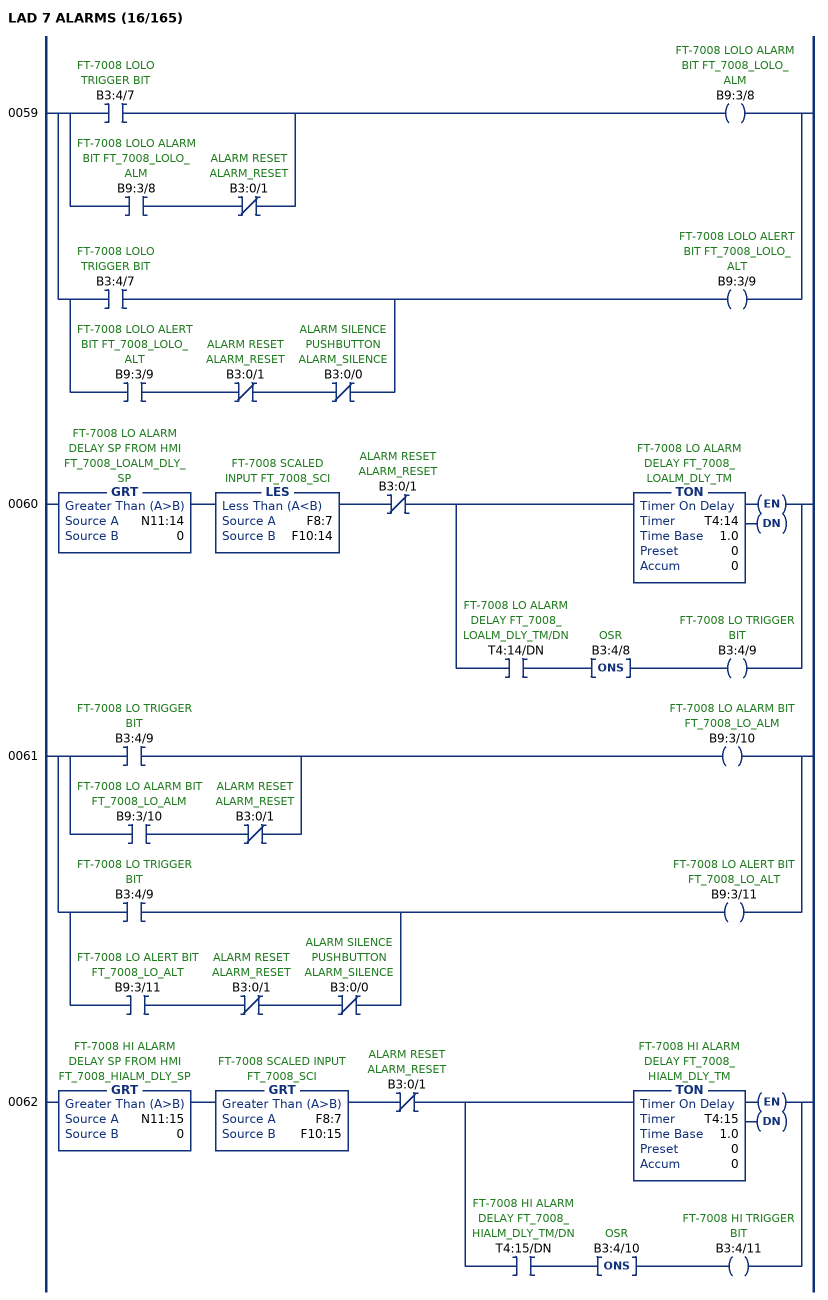
% Rung: 59 %
SOR BST BST XIC B3:4/7 NXB XIC B9:3/8 XIO B3:0/1 BND OTE B9:3/8 NXB BST XIC B3:4/7 NXB XIC B9:3/9 XIO B3:0/1 XIO B3:0/0 BND OTE B9:3/9 BND EOR
%   B3:4/7  "FT-7008 LOLO TRIGGER BIT" %
%   B9:3/8  FT_7008_LOLO_ALM  "FT-7008 LOLO ALARM BIT" %
%   B3:0/1  ALARM_RESET  "ALARM RESET" %
%   B9:3/9  FT_7008_LOLO_ALT  "FT-7008 LOLO ALERT BIT" %
%   B3:0/0  ALARM_SILENCE  "ALARM SILENCE PUSHBUTTON" %
% Rung: 60 %
SOR GRT N11:14 0 LES F8:7 F10:14 XIO B3:0/1 BST TON T4:14 1.0 0 0 NXB XIC T4:14/DN OSR B3:4/8 OTE B3:4/9 BND EOR
%   N11:14  FT_7008_LOALM_DLY_SP  "FT-7008 LO ALARM DELAY SP FROM HMI" %
%   F8:7  FT_7008_SCI  "FT-7008 SCALED INPUT" %
%   F10:14  FT_7008_LOALM_SP  "FT-7008 LO ALARM SP" %
%   B3:0/1  ALARM_RESET  "ALARM RESET" %
%   T4:14  FT_7008_LOALM_DLY_TM  "FT-7008 LO ALARM DELAY" %
%   B3:4/8  "OSR" %
%   B3:4/9  "FT-7008 LO TRIGGER BIT" %
% Rung: 61 %
SOR BST BST XIC B3:4/9 NXB XIC B9:3/10 XIO B3:0/1 BND OTE B9:3/10 NXB BST XIC B3:4/9 NXB XIC B9:3/11 XIO B3:0/1 XIO B3:0/0 BND OTE B9:3/11 BND EOR
%   B3:4/9  "FT-7008 LO TRIGGER BIT" %
%   B9:3/10  FT_7008_LO_ALM  "FT-7008 LO ALARM BIT" %
%   B3:0/1  ALARM_RESET  "ALARM RESET" %
%   B9:3/11  FT_7008_LO_ALT  "FT-7008 LO ALERT BIT" %
%   B3:0/0  ALARM_SILENCE  "ALARM SILENCE PUSHBUTTON" %
% Rung: 62 %
SOR GRT N11:15 0 GRT F8:7 F10:15 XIO B3:0/1 BST TON T4:15 1.0 0 0 NXB XIC T4:15/DN OSR B3:4/10 OTE B3:4/11 BND EOR
%   N11:15  FT_7008_HIALM_DLY_SP  "FT-7008 HI ALARM DELAY SP FROM HMI" %
%   F8:7  FT_7008_SCI  "FT-7008 SCALED INPUT" %
%   F10:15  FT_7008_HIALM_SP  "FT-7008 HI ALARM SP" %
%   B3:0/1  ALARM_RESET  "ALARM RESET" %
%   T4:15  FT_7008_HIALM_DLY_TM  "FT-7008 HI ALARM DELAY" %
%   B3:4/10  "OSR" %
%   B3:4/11  "FT-7008 HI TRIGGER BIT" %

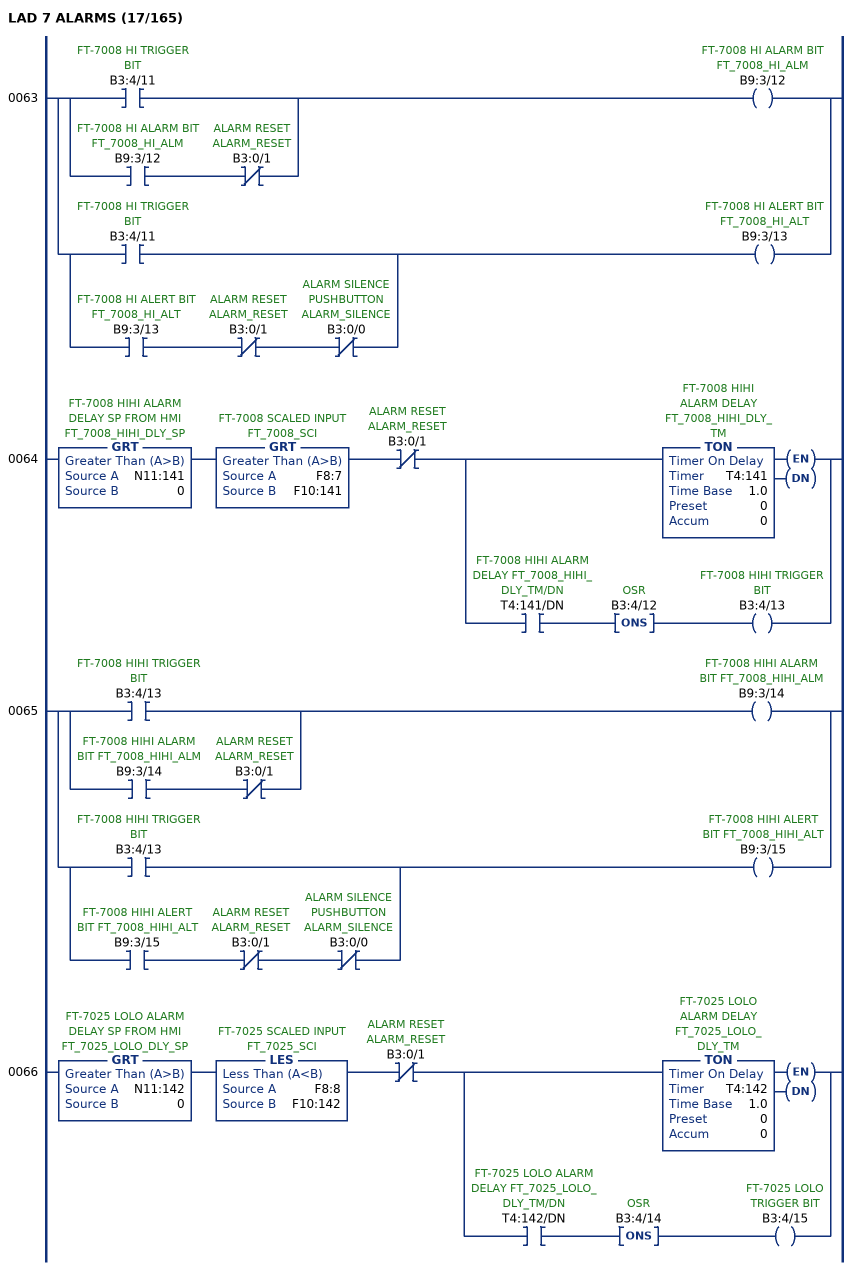
% Rung: 63 %
SOR BST BST XIC B3:4/11 NXB XIC B9:3/12 XIO B3:0/1 BND OTE B9:3/12 NXB BST XIC B3:4/11 NXB XIC B9:3/13 XIO B3:0/1 XIO B3:0/0 BND OTE B9:3/13 BND EOR
%   B3:4/11  "FT-7008 HI TRIGGER BIT" %
%   B9:3/12  FT_7008_HI_ALM  "FT-7008 HI ALARM BIT" %
%   B3:0/1  ALARM_RESET  "ALARM RESET" %
%   B9:3/13  FT_7008_HI_ALT  "FT-7008 HI ALERT BIT" %
%   B3:0/0  ALARM_SILENCE  "ALARM SILENCE PUSHBUTTON" %
% Rung: 64 %
SOR GRT N11:141 0 GRT F8:7 F10:141 XIO B3:0/1 BST TON T4:141 1.0 0 0 NXB XIC T4:141/DN OSR B3:4/12 OTE B3:4/13 BND EOR
%   N11:141  FT_7008_HIHI_DLY_SP  "FT-7008 HIHI ALARM DELAY SP FROM HMI" %
%   F8:7  FT_7008_SCI  "FT-7008 SCALED INPUT" %
%   F10:141  FT_7008_HIHI_SP  "FT-7008 HIHI ALARM SP" %
%   B3:0/1  ALARM_RESET  "ALARM RESET" %
%   T4:141  FT_7008_HIHI_DLY_TM  "FT-7008 HIHI ALARM DELAY" %
%   B3:4/12  "OSR" %
%   B3:4/13  "FT-7008 HIHI TRIGGER BIT" %
% Rung: 65 %
SOR BST BST XIC B3:4/13 NXB XIC B9:3/14 XIO B3:0/1 BND OTE B9:3/14 NXB BST XIC B3:4/13 NXB XIC B9:3/15 XIO B3:0/1 XIO B3:0/0 BND OTE B9:3/15 BND EOR
%   B3:4/13  "FT-7008 HIHI TRIGGER BIT" %
%   B9:3/14  FT_7008_HIHI_ALM  "FT-7008 HIHI ALARM BIT" %
%   B3:0/1  ALARM_RESET  "ALARM RESET" %
%   B9:3/15  FT_7008_HIHI_ALT  "FT-7008 HIHI ALERT BIT" %
%   B3:0/0  ALARM_SILENCE  "ALARM SILENCE PUSHBUTTON" %
% Rung: 66 %
SOR GRT N11:142 0 LES F8:8 F10:142 XIO B3:0/1 BST TON T4:142 1.0 0 0 NXB XIC T4:142/DN OSR B3:4/14 OTE B3:4/15 BND EOR
%   N11:142  FT_7025_LOLO_DLY_SP  "FT-7025 LOLO ALARM DELAY SP FROM HMI" %
%   F8:8  FT_7025_SCI  "FT-7025 SCALED INPUT" %
%   F10:142  FT_7025_LOLO_SP  "FT-7025 LOLO ALARM SP" %
%   B3:0/1  ALARM_RESET  "ALARM RESET" %
%   T4:142  FT_7025_LOLO_DLY_TM  "FT-7025 LOLO ALARM DELAY" %
%   B3:4/14  "OSR" %
%   B3:4/15  "FT-7025 LOLO TRIGGER BIT" %

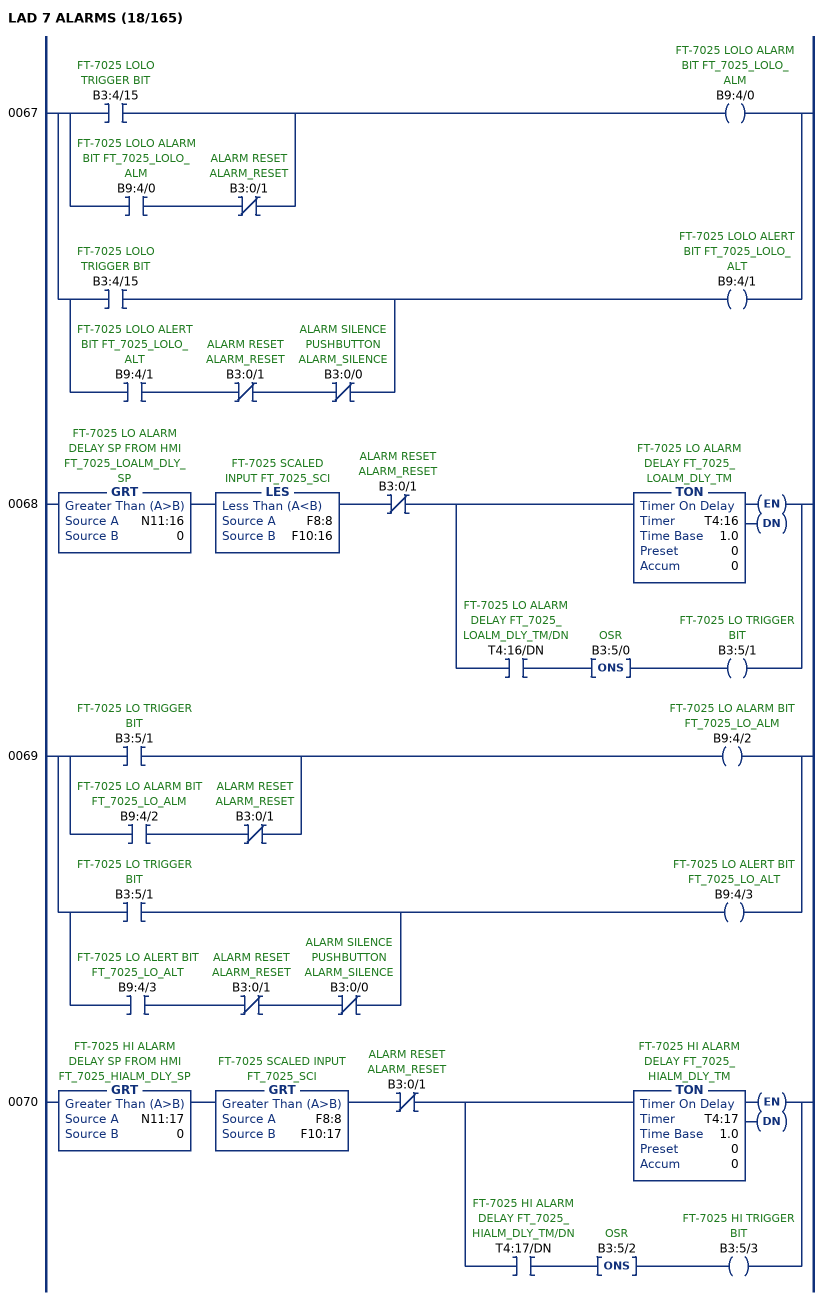
% Rung: 67 %
SOR BST BST XIC B3:4/15 NXB XIC B9:4/0 XIO B3:0/1 BND OTE B9:4/0 NXB BST XIC B3:4/15 NXB XIC B9:4/1 XIO B3:0/1 XIO B3:0/0 BND OTE B9:4/1 BND EOR
%   B3:4/15  "FT-7025 LOLO TRIGGER BIT" %
%   B9:4/0  FT_7025_LOLO_ALM  "FT-7025 LOLO ALARM BIT" %
%   B3:0/1  ALARM_RESET  "ALARM RESET" %
%   B9:4/1  FT_7025_LOLO_ALT  "FT-7025 LOLO ALERT BIT" %
%   B3:0/0  ALARM_SILENCE  "ALARM SILENCE PUSHBUTTON" %
% Rung: 68 %
SOR GRT N11:16 0 LES F8:8 F10:16 XIO B3:0/1 BST TON T4:16 1.0 0 0 NXB XIC T4:16/DN OSR B3:5/0 OTE B3:5/1 BND EOR
%   N11:16  FT_7025_LOALM_DLY_SP  "FT-7025 LO ALARM DELAY SP FROM HMI" %
%   F8:8  FT_7025_SCI  "FT-7025 SCALED INPUT" %
%   F10:16  FT_7025_LOALM_SP  "FT-7025 LO ALARM SP" %
%   B3:0/1  ALARM_RESET  "ALARM RESET" %
%   T4:16  FT_7025_LOALM_DLY_TM  "FT-7025 LO ALARM DELAY" %
%   B3:5/0  "OSR" %
%   B3:5/1  "FT-7025 LO TRIGGER BIT" %
% Rung: 69 %
SOR BST BST XIC B3:5/1 NXB XIC B9:4/2 XIO B3:0/1 BND OTE B9:4/2 NXB BST XIC B3:5/1 NXB XIC B9:4/3 XIO B3:0/1 XIO B3:0/0 BND OTE B9:4/3 BND EOR
%   B3:5/1  "FT-7025 LO TRIGGER BIT" %
%   B9:4/2  FT_7025_LO_ALM  "FT-7025 LO ALARM BIT" %
%   B3:0/1  ALARM_RESET  "ALARM RESET" %
%   B9:4/3  FT_7025_LO_ALT  "FT-7025 LO ALERT BIT" %
%   B3:0/0  ALARM_SILENCE  "ALARM SILENCE PUSHBUTTON" %
% Rung: 70 %
SOR GRT N11:17 0 GRT F8:8 F10:17 XIO B3:0/1 BST TON T4:17 1.0 0 0 NXB XIC T4:17/DN OSR B3:5/2 OTE B3:5/3 BND EOR
%   N11:17  FT_7025_HIALM_DLY_SP  "FT-7025 HI ALARM DELAY SP FROM HMI" %
%   F8:8  FT_7025_SCI  "FT-7025 SCALED INPUT" %
%   F10:17  FT_7025_HIALM_SP  "FT-7025 HI ALARM SP" %
%   B3:0/1  ALARM_RESET  "ALARM RESET" %
%   T4:17  FT_7025_HIALM_DLY_TM  "FT-7025 HI ALARM DELAY" %
%   B3:5/2  "OSR" %
%   B3:5/3  "FT-7025 HI TRIGGER BIT" %

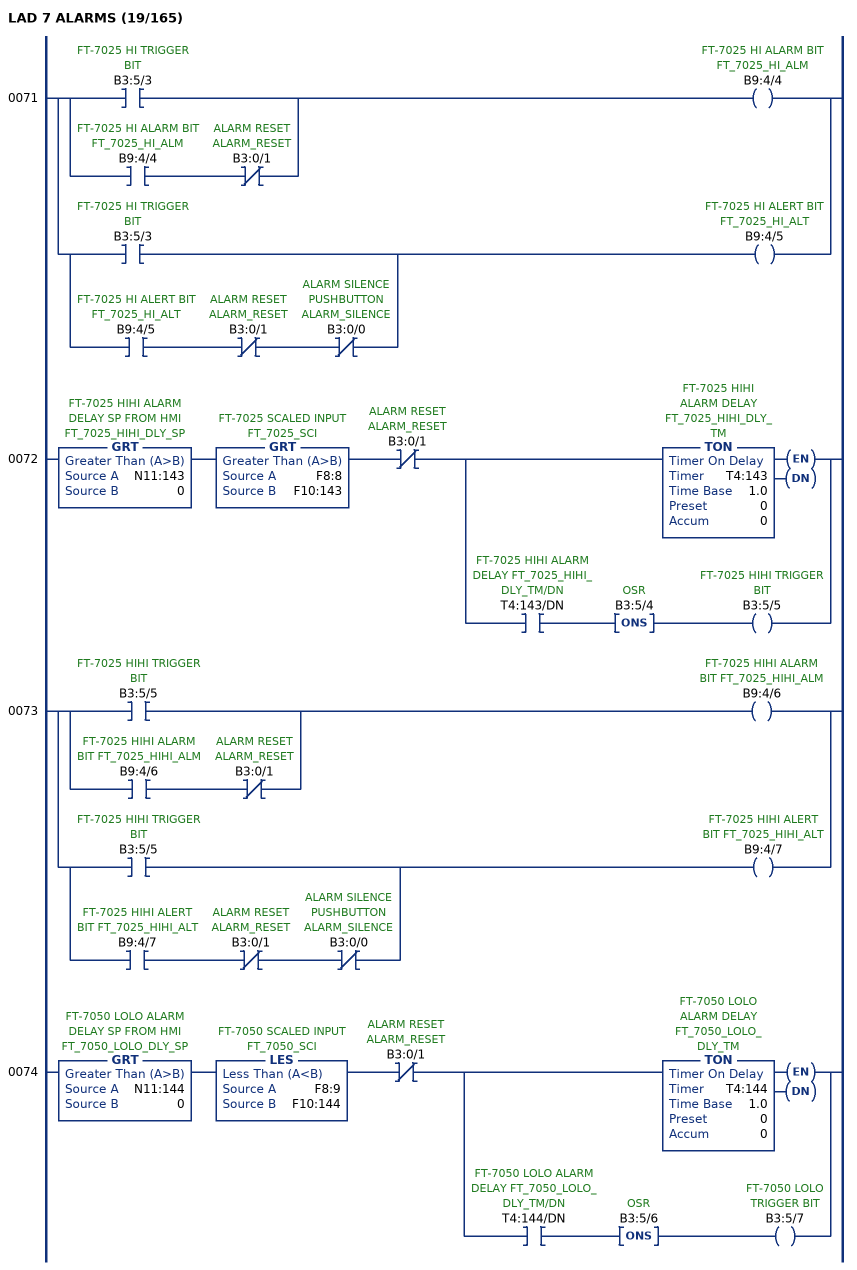
% Rung: 71 %
SOR BST BST XIC B3:5/3 NXB XIC B9:4/4 XIO B3:0/1 BND OTE B9:4/4 NXB BST XIC B3:5/3 NXB XIC B9:4/5 XIO B3:0/1 XIO B3:0/0 BND OTE B9:4/5 BND EOR
%   B3:5/3  "FT-7025 HI TRIGGER BIT" %
%   B9:4/4  FT_7025_HI_ALM  "FT-7025 HI ALARM BIT" %
%   B3:0/1  ALARM_RESET  "ALARM RESET" %
%   B9:4/5  FT_7025_HI_ALT  "FT-7025 HI ALERT BIT" %
%   B3:0/0  ALARM_SILENCE  "ALARM SILENCE PUSHBUTTON" %
% Rung: 72 %
SOR GRT N11:143 0 GRT F8:8 F10:143 XIO B3:0/1 BST TON T4:143 1.0 0 0 NXB XIC T4:143/DN OSR B3:5/4 OTE B3:5/5 BND EOR
%   N11:143  FT_7025_HIHI_DLY_SP  "FT-7025 HIHI ALARM DELAY SP FROM HMI" %
%   F8:8  FT_7025_SCI  "FT-7025 SCALED INPUT" %
%   F10:143  FT_7025_HIHI_SP  "FT-7025 HIHI ALARM SP" %
%   B3:0/1  ALARM_RESET  "ALARM RESET" %
%   T4:143  FT_7025_HIHI_DLY_TM  "FT-7025 HIHI ALARM DELAY" %
%   B3:5/4  "OSR" %
%   B3:5/5  "FT-7025 HIHI TRIGGER BIT" %
% Rung: 73 %
SOR BST BST XIC B3:5/5 NXB XIC B9:4/6 XIO B3:0/1 BND OTE B9:4/6 NXB BST XIC B3:5/5 NXB XIC B9:4/7 XIO B3:0/1 XIO B3:0/0 BND OTE B9:4/7 BND EOR
%   B3:5/5  "FT-7025 HIHI TRIGGER BIT" %
%   B9:4/6  FT_7025_HIHI_ALM  "FT-7025 HIHI ALARM BIT" %
%   B3:0/1  ALARM_RESET  "ALARM RESET" %
%   B9:4/7  FT_7025_HIHI_ALT  "FT-7025 HIHI ALERT BIT" %
%   B3:0/0  ALARM_SILENCE  "ALARM SILENCE PUSHBUTTON" %
% Rung: 74 %
SOR GRT N11:144 0 LES F8:9 F10:144 XIO B3:0/1 BST TON T4:144 1.0 0 0 NXB XIC T4:144/DN OSR B3:5/6 OTE B3:5/7 BND EOR
%   N11:144  FT_7050_LOLO_DLY_SP  "FT-7050 LOLO ALARM DELAY SP FROM HMI" %
%   F8:9  FT_7050_SCI  "FT-7050 SCALED INPUT" %
%   F10:144  FT_7050_LOLO_SP  "FT-7050 LOLO ALARM SP" %
%   B3:0/1  ALARM_RESET  "ALARM RESET" %
%   T4:144  FT_7050_LOLO_DLY_TM  "FT-7050 LOLO ALARM DELAY" %
%   B3:5/6  "OSR" %
%   B3:5/7  "FT-7050 LOLO TRIGGER BIT" %

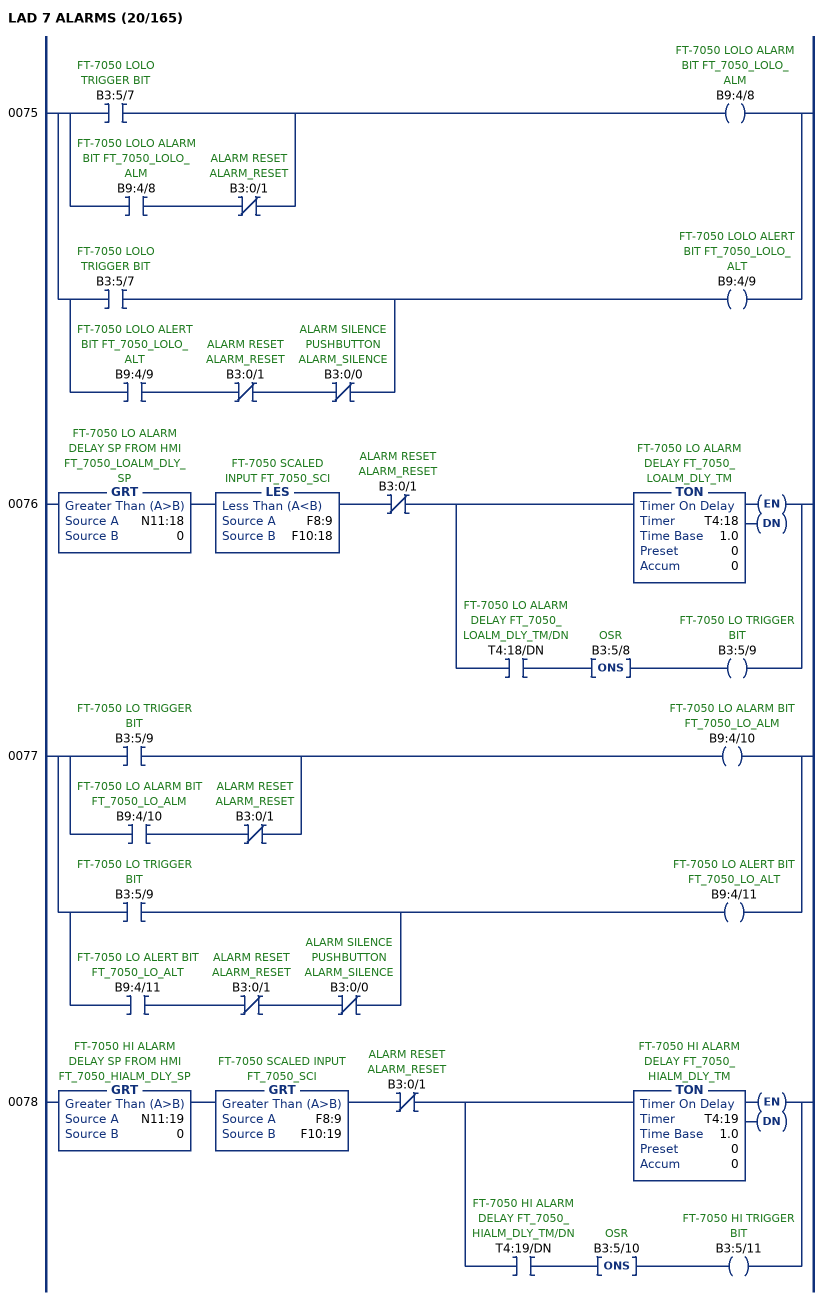
% Rung: 75 %
SOR BST BST XIC B3:5/7 NXB XIC B9:4/8 XIO B3:0/1 BND OTE B9:4/8 NXB BST XIC B3:5/7 NXB XIC B9:4/9 XIO B3:0/1 XIO B3:0/0 BND OTE B9:4/9 BND EOR
%   B3:5/7  "FT-7050 LOLO TRIGGER BIT" %
%   B9:4/8  FT_7050_LOLO_ALM  "FT-7050 LOLO ALARM BIT" %
%   B3:0/1  ALARM_RESET  "ALARM RESET" %
%   B9:4/9  FT_7050_LOLO_ALT  "FT-7050 LOLO ALERT BIT" %
%   B3:0/0  ALARM_SILENCE  "ALARM SILENCE PUSHBUTTON" %
% Rung: 76 %
SOR GRT N11:18 0 LES F8:9 F10:18 XIO B3:0/1 BST TON T4:18 1.0 0 0 NXB XIC T4:18/DN OSR B3:5/8 OTE B3:5/9 BND EOR
%   N11:18  FT_7050_LOALM_DLY_SP  "FT-7050 LO ALARM DELAY SP FROM HMI" %
%   F8:9  FT_7050_SCI  "FT-7050 SCALED INPUT" %
%   F10:18  FT_7050_LOALM_SP  "FT-7050 LO ALARM SP" %
%   B3:0/1  ALARM_RESET  "ALARM RESET" %
%   T4:18  FT_7050_LOALM_DLY_TM  "FT-7050 LO ALARM DELAY" %
%   B3:5/8  "OSR" %
%   B3:5/9  "FT-7050 LO TRIGGER BIT" %
% Rung: 77 %
SOR BST BST XIC B3:5/9 NXB XIC B9:4/10 XIO B3:0/1 BND OTE B9:4/10 NXB BST XIC B3:5/9 NXB XIC B9:4/11 XIO B3:0/1 XIO B3:0/0 BND OTE B9:4/11 BND EOR
%   B3:5/9  "FT-7050 LO TRIGGER BIT" %
%   B9:4/10  FT_7050_LO_ALM  "FT-7050 LO ALARM BIT" %
%   B3:0/1  ALARM_RESET  "ALARM RESET" %
%   B9:4/11  FT_7050_LO_ALT  "FT-7050 LO ALERT BIT" %
%   B3:0/0  ALARM_SILENCE  "ALARM SILENCE PUSHBUTTON" %
% Rung: 78 %
SOR GRT N11:19 0 GRT F8:9 F10:19 XIO B3:0/1 BST TON T4:19 1.0 0 0 NXB XIC T4:19/DN OSR B3:5/10 OTE B3:5/11 BND EOR
%   N11:19  FT_7050_HIALM_DLY_SP  "FT-7050 HI ALARM DELAY SP FROM HMI" %
%   F8:9  FT_7050_SCI  "FT-7050 SCALED INPUT" %
%   F10:19  FT_7050_HIALM_SP  "FT-7050 HI ALARM SP" %
%   B3:0/1  ALARM_RESET  "ALARM RESET" %
%   T4:19  FT_7050_HIALM_DLY_TM  "FT-7050 HI ALARM DELAY" %
%   B3:5/10  "OSR" %
%   B3:5/11  "FT-7050 HI TRIGGER BIT" %

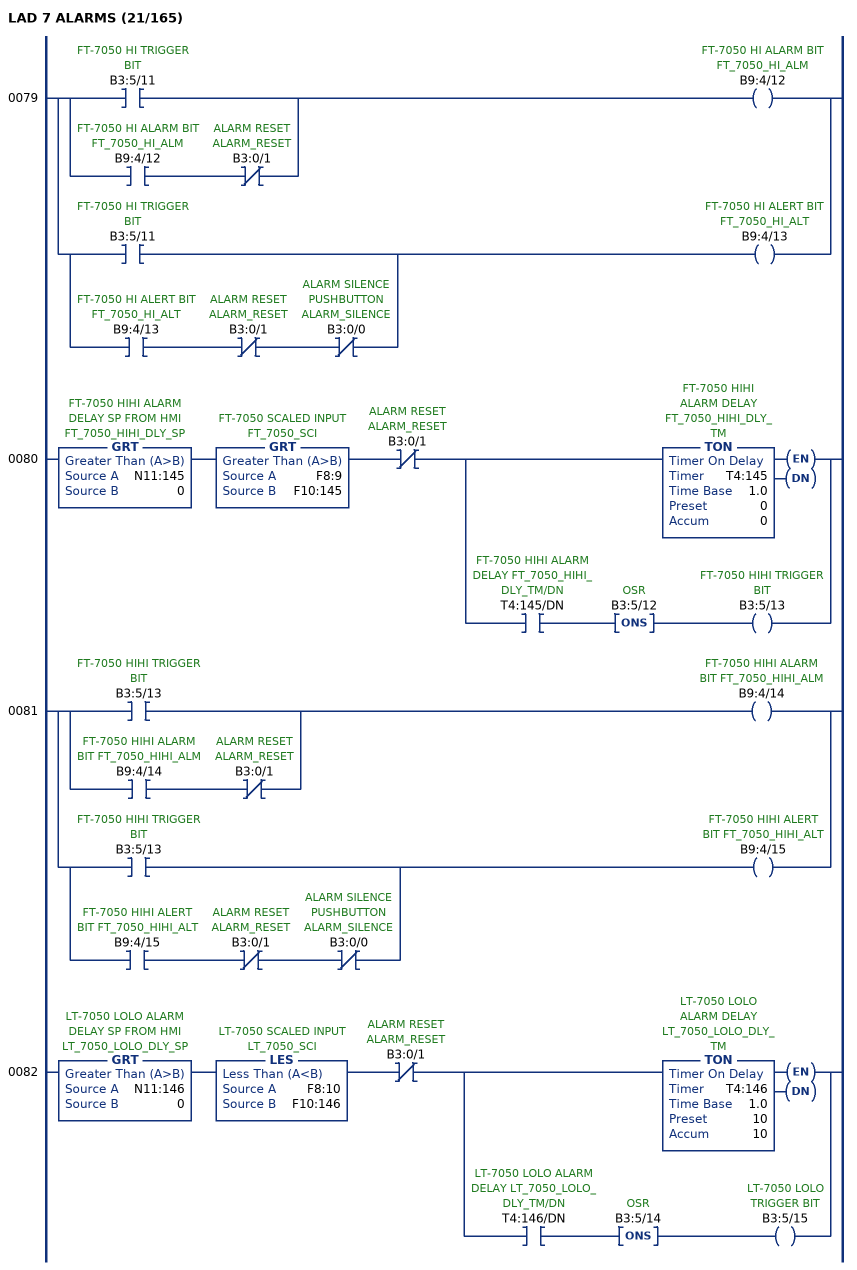
% Rung: 79 %
SOR BST BST XIC B3:5/11 NXB XIC B9:4/12 XIO B3:0/1 BND OTE B9:4/12 NXB BST XIC B3:5/11 NXB XIC B9:4/13 XIO B3:0/1 XIO B3:0/0 BND OTE B9:4/13 BND EOR
%   B3:5/11  "FT-7050 HI TRIGGER BIT" %
%   B9:4/12  FT_7050_HI_ALM  "FT-7050 HI ALARM BIT" %
%   B3:0/1  ALARM_RESET  "ALARM RESET" %
%   B9:4/13  FT_7050_HI_ALT  "FT-7050 HI ALERT BIT" %
%   B3:0/0  ALARM_SILENCE  "ALARM SILENCE PUSHBUTTON" %
% Rung: 80 %
SOR GRT N11:145 0 GRT F8:9 F10:145 XIO B3:0/1 BST TON T4:145 1.0 0 0 NXB XIC T4:145/DN OSR B3:5/12 OTE B3:5/13 BND EOR
%   N11:145  FT_7050_HIHI_DLY_SP  "FT-7050 HIHI ALARM DELAY SP FROM HMI" %
%   F8:9  FT_7050_SCI  "FT-7050 SCALED INPUT" %
%   F10:145  FT_7050_HIHI_SP  "FT-7050 HIHI ALARM SP" %
%   B3:0/1  ALARM_RESET  "ALARM RESET" %
%   T4:145  FT_7050_HIHI_DLY_TM  "FT-7050 HIHI ALARM DELAY" %
%   B3:5/12  "OSR" %
%   B3:5/13  "FT-7050 HIHI TRIGGER BIT" %
% Rung: 81 %
SOR BST BST XIC B3:5/13 NXB XIC B9:4/14 XIO B3:0/1 BND OTE B9:4/14 NXB BST XIC B3:5/13 NXB XIC B9:4/15 XIO B3:0/1 XIO B3:0/0 BND OTE B9:4/15 BND EOR
%   B3:5/13  "FT-7050 HIHI TRIGGER BIT" %
%   B9:4/14  FT_7050_HIHI_ALM  "FT-7050 HIHI ALARM BIT" %
%   B3:0/1  ALARM_RESET  "ALARM RESET" %
%   B9:4/15  FT_7050_HIHI_ALT  "FT-7050 HIHI ALERT BIT" %
%   B3:0/0  ALARM_SILENCE  "ALARM SILENCE PUSHBUTTON" %
% Rung: 82 %
SOR GRT N11:146 0 LES F8:10 F10:146 XIO B3:0/1 BST TON T4:146 1.0 10 10 NXB XIC T4:146/DN OSR B3:5/14 OTE B3:5/15 BND EOR
%   N11:146  LT_7050_LOLO_DLY_SP  "LT-7050 LOLO ALARM DELAY SP FROM HMI" %
%   F8:10  LT_7050_SCI  "LT-7050 SCALED INPUT" %
%   F10:146  LT_7050_LOLO_SP  "LT-7050 LOLO ALARM SP" %
%   B3:0/1  ALARM_RESET  "ALARM RESET" %
%   T4:146  LT_7050_LOLO_DLY_TM  "LT-7050 LOLO ALARM DELAY" %
%   B3:5/14  "OSR" %
%   B3:5/15  "LT-7050 LOLO TRIGGER BIT" %

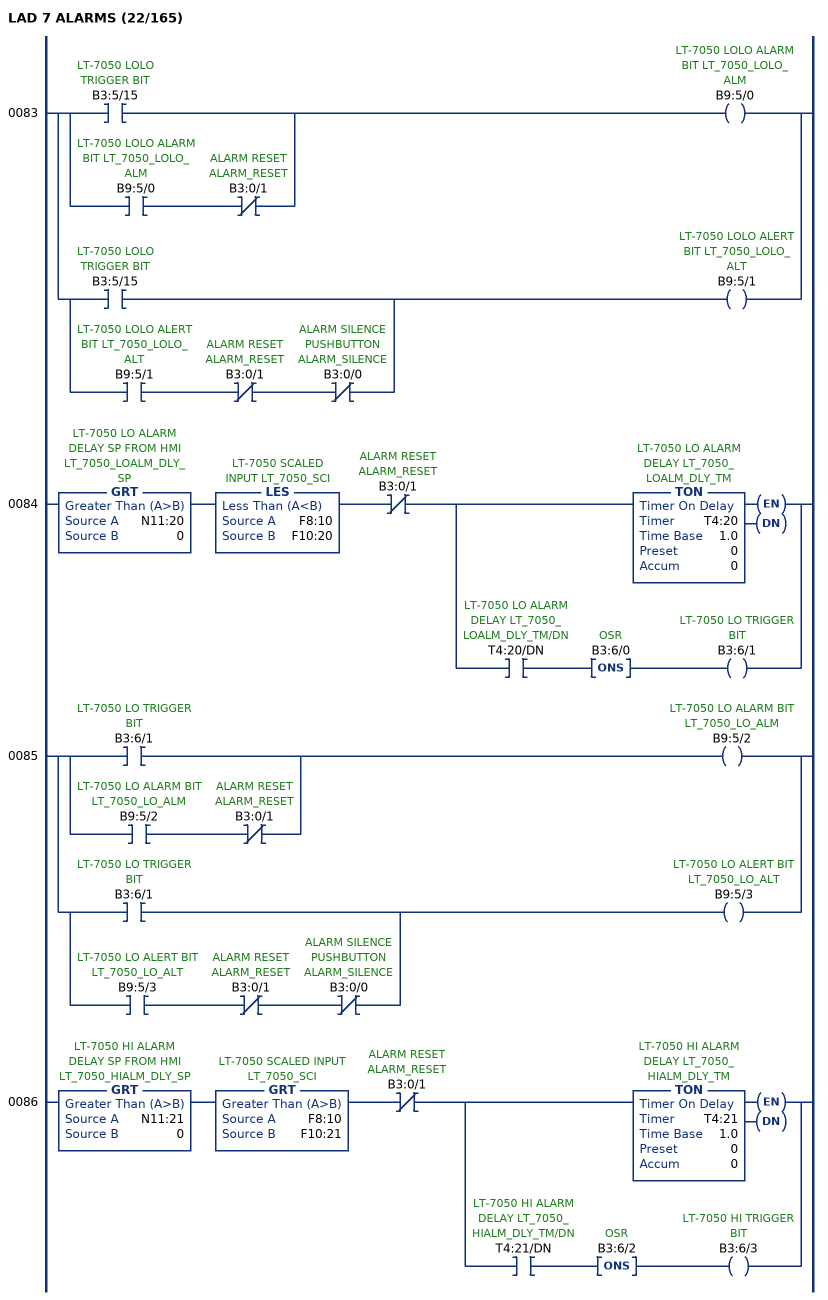
% Rung: 83 %
SOR BST BST XIC B3:5/15 NXB XIC B9:5/0 XIO B3:0/1 BND OTE B9:5/0 NXB BST XIC B3:5/15 NXB XIC B9:5/1 XIO B3:0/1 XIO B3:0/0 BND OTE B9:5/1 BND EOR
%   B3:5/15  "LT-7050 LOLO TRIGGER BIT" %
%   B9:5/0  LT_7050_LOLO_ALM  "LT-7050 LOLO ALARM BIT" %
%   B3:0/1  ALARM_RESET  "ALARM RESET" %
%   B9:5/1  LT_7050_LOLO_ALT  "LT-7050 LOLO ALERT BIT" %
%   B3:0/0  ALARM_SILENCE  "ALARM SILENCE PUSHBUTTON" %
% Rung: 84 %
SOR GRT N11:20 0 LES F8:10 F10:20 XIO B3:0/1 BST TON T4:20 1.0 0 0 NXB XIC T4:20/DN OSR B3:6/0 OTE B3:6/1 BND EOR
%   N11:20  LT_7050_LOALM_DLY_SP  "LT-7050 LO ALARM DELAY SP FROM HMI" %
%   F8:10  LT_7050_SCI  "LT-7050 SCALED INPUT" %
%   F10:20  LT_7050_LOALM_SP  "LT-7050 LO ALARM SP" %
%   B3:0/1  ALARM_RESET  "ALARM RESET" %
%   T4:20  LT_7050_LOALM_DLY_TM  "LT-7050 LO ALARM DELAY" %
%   B3:6/0  "OSR" %
%   B3:6/1  "LT-7050 LO TRIGGER BIT" %
% Rung: 85 %
SOR BST BST XIC B3:6/1 NXB XIC B9:5/2 XIO B3:0/1 BND OTE B9:5/2 NXB BST XIC B3:6/1 NXB XIC B9:5/3 XIO B3:0/1 XIO B3:0/0 BND OTE B9:5/3 BND EOR
%   B3:6/1  "LT-7050 LO TRIGGER BIT" %
%   B9:5/2  LT_7050_LO_ALM  "LT-7050 LO ALARM BIT" %
%   B3:0/1  ALARM_RESET  "ALARM RESET" %
%   B9:5/3  LT_7050_LO_ALT  "LT-7050 LO ALERT BIT" %
%   B3:0/0  ALARM_SILENCE  "ALARM SILENCE PUSHBUTTON" %
% Rung: 86 %
SOR GRT N11:21 0 GRT F8:10 F10:21 XIO B3:0/1 BST TON T4:21 1.0 0 0 NXB XIC T4:21/DN OSR B3:6/2 OTE B3:6/3 BND EOR
%   N11:21  LT_7050_HIALM_DLY_SP  "LT-7050 HI ALARM DELAY SP FROM HMI" %
%   F8:10  LT_7050_SCI  "LT-7050 SCALED INPUT" %
%   F10:21  LT_7050_HIALM_SP  "LT-7050 HI ALARM SP" %
%   B3:0/1  ALARM_RESET  "ALARM RESET" %
%   T4:21  LT_7050_HIALM_DLY_TM  "LT-7050 HI ALARM DELAY" %
%   B3:6/2  "OSR" %
%   B3:6/3  "LT-7050 HI TRIGGER BIT" %

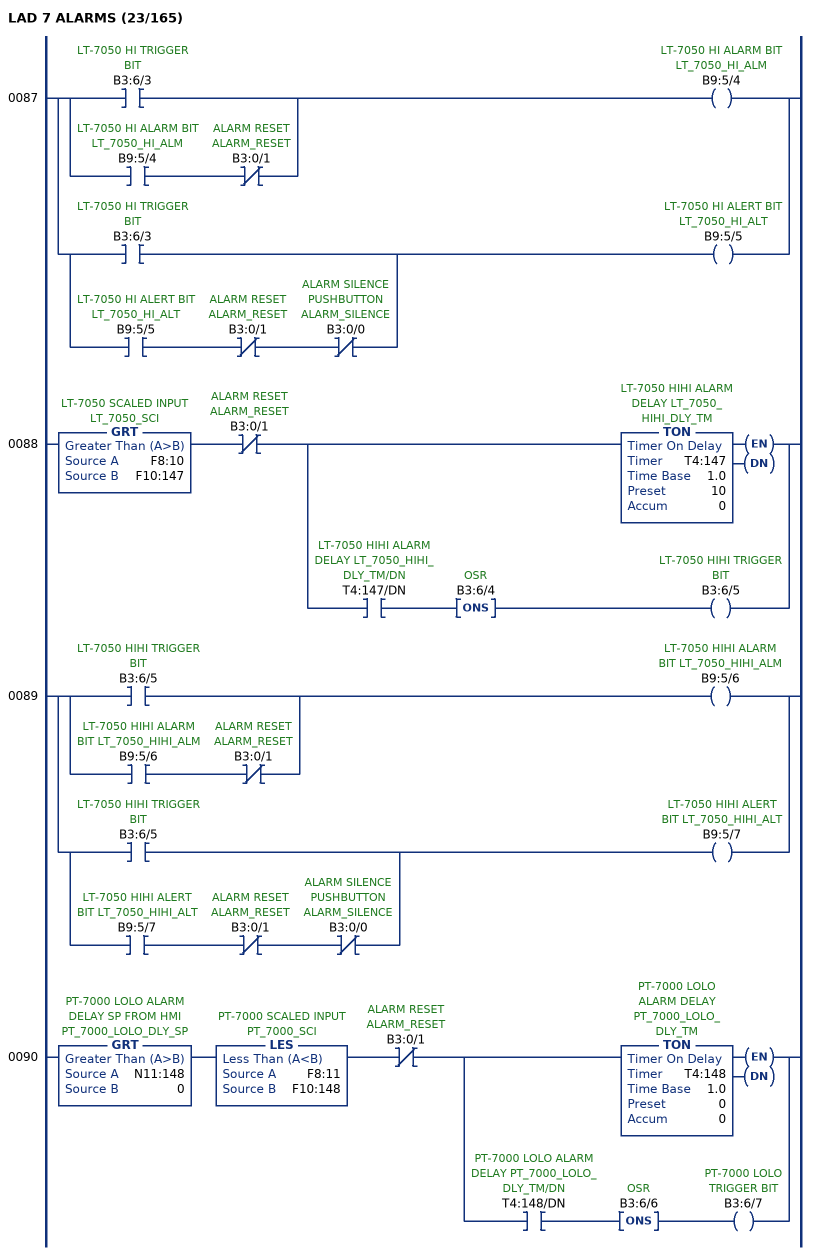
% Rung: 87 %
SOR BST BST XIC B3:6/3 NXB XIC B9:5/4 XIO B3:0/1 BND OTE B9:5/4 NXB BST XIC B3:6/3 NXB XIC B9:5/5 XIO B3:0/1 XIO B3:0/0 BND OTE B9:5/5 BND EOR
%   B3:6/3  "LT-7050 HI TRIGGER BIT" %
%   B9:5/4  LT_7050_HI_ALM  "LT-7050 HI ALARM BIT" %
%   B3:0/1  ALARM_RESET  "ALARM RESET" %
%   B9:5/5  LT_7050_HI_ALT  "LT-7050 HI ALERT BIT" %
%   B3:0/0  ALARM_SILENCE  "ALARM SILENCE PUSHBUTTON" %
% Rung: 88 %
SOR GRT F8:10 F10:147 XIO B3:0/1 BST TON T4:147 1.0 10 0 NXB XIC T4:147/DN OSR B3:6/4 OTE B3:6/5 BND EOR
%   F8:10  LT_7050_SCI  "LT-7050 SCALED INPUT" %
%   F10:147  LT_7050_HIHI_SP  "LT-7050 HIHI ALARM SP" %
%   B3:0/1  ALARM_RESET  "ALARM RESET" %
%   T4:147  LT_7050_HIHI_DLY_TM  "LT-7050 HIHI ALARM DELAY" %
%   B3:6/4  "OSR" %
%   B3:6/5  "LT-7050 HIHI TRIGGER BIT" %
% Rung: 89 %
SOR BST BST XIC B3:6/5 NXB XIC B9:5/6 XIO B3:0/1 BND OTE B9:5/6 NXB BST XIC B3:6/5 NXB XIC B9:5/7 XIO B3:0/1 XIO B3:0/0 BND OTE B9:5/7 BND EOR
%   B3:6/5  "LT-7050 HIHI TRIGGER BIT" %
%   B9:5/6  LT_7050_HIHI_ALM  "LT-7050 HIHI ALARM BIT" %
%   B3:0/1  ALARM_RESET  "ALARM RESET" %
%   B9:5/7  LT_7050_HIHI_ALT  "LT-7050 HIHI ALERT BIT" %
%   B3:0/0  ALARM_SILENCE  "ALARM SILENCE PUSHBUTTON" %
% Rung: 90 %
SOR GRT N11:148 0 LES F8:11 F10:148 XIO B3:0/1 BST TON T4:148 1.0 0 0 NXB XIC T4:148/DN OSR B3:6/6 OTE B3:6/7 BND EOR
%   N11:148  PT_7000_LOLO_DLY_SP  "PT-7000 LOLO ALARM DELAY SP FROM HMI" %
%   F8:11  PT_7000_SCI  "PT-7000 SCALED INPUT" %
%   F10:148  PT_7000_LOLO_SP  "PT-7000 LOLO ALARM SP" %
%   B3:0/1  ALARM_RESET  "ALARM RESET" %
%   T4:148  PT_7000_LOLO_DLY_TM  "PT-7000 LOLO ALARM DELAY" %
%   B3:6/6  "OSR" %
%   B3:6/7  "PT-7000 LOLO TRIGGER BIT" %

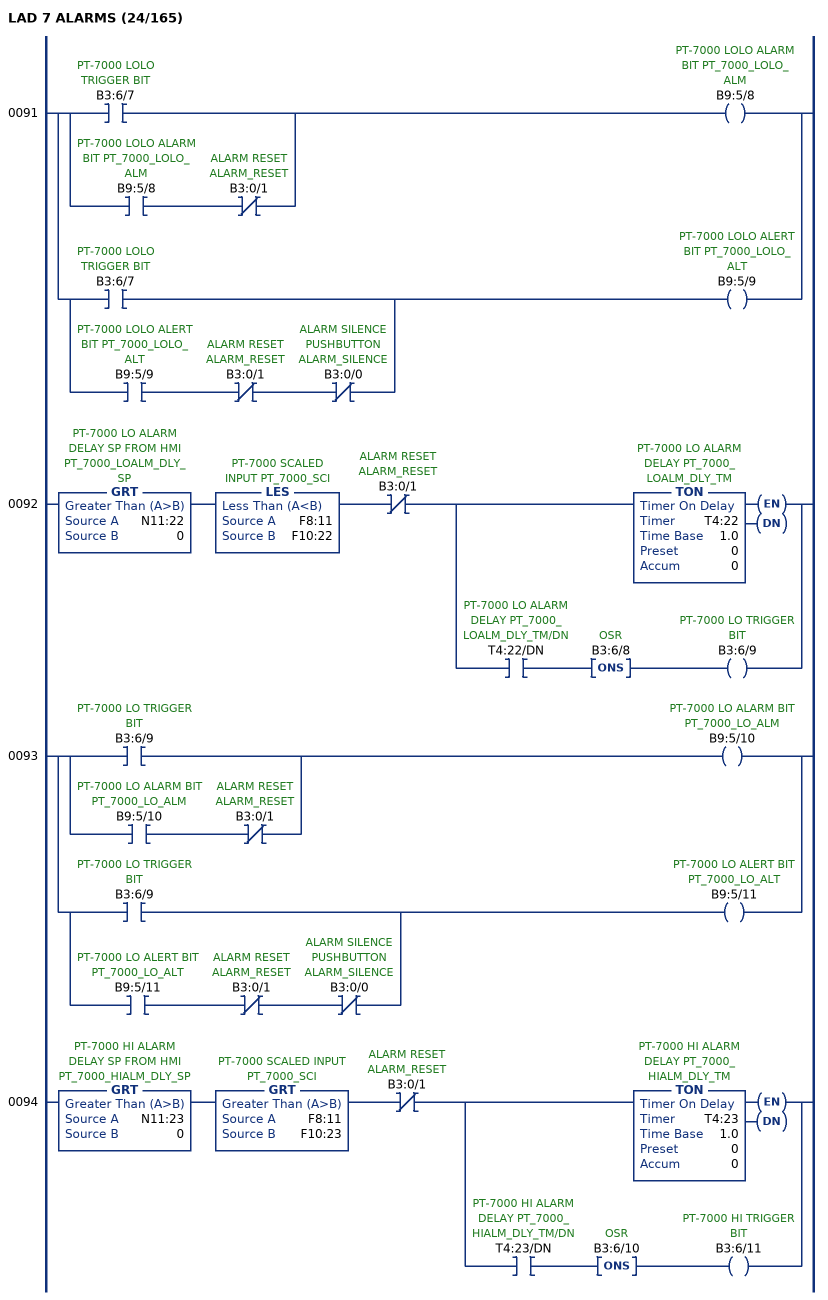
% Rung: 91 %
SOR BST BST XIC B3:6/7 NXB XIC B9:5/8 XIO B3:0/1 BND OTE B9:5/8 NXB BST XIC B3:6/7 NXB XIC B9:5/9 XIO B3:0/1 XIO B3:0/0 BND OTE B9:5/9 BND EOR
%   B3:6/7  "PT-7000 LOLO TRIGGER BIT" %
%   B9:5/8  PT_7000_LOLO_ALM  "PT-7000 LOLO ALARM BIT" %
%   B3:0/1  ALARM_RESET  "ALARM RESET" %
%   B9:5/9  PT_7000_LOLO_ALT  "PT-7000 LOLO ALERT BIT" %
%   B3:0/0  ALARM_SILENCE  "ALARM SILENCE PUSHBUTTON" %
% Rung: 92 %
SOR GRT N11:22 0 LES F8:11 F10:22 XIO B3:0/1 BST TON T4:22 1.0 0 0 NXB XIC T4:22/DN OSR B3:6/8 OTE B3:6/9 BND EOR
%   N11:22  PT_7000_LOALM_DLY_SP  "PT-7000 LO ALARM DELAY SP FROM HMI" %
%   F8:11  PT_7000_SCI  "PT-7000 SCALED INPUT" %
%   F10:22  PT_7000_LOALM_SP  "PT-7000 LO ALARM SP" %
%   B3:0/1  ALARM_RESET  "ALARM RESET" %
%   T4:22  PT_7000_LOALM_DLY_TM  "PT-7000 LO ALARM DELAY" %
%   B3:6/8  "OSR" %
%   B3:6/9  "PT-7000 LO TRIGGER BIT" %
% Rung: 93 %
SOR BST BST XIC B3:6/9 NXB XIC B9:5/10 XIO B3:0/1 BND OTE B9:5/10 NXB BST XIC B3:6/9 NXB XIC B9:5/11 XIO B3:0/1 XIO B3:0/0 BND OTE B9:5/11 BND EOR
%   B3:6/9  "PT-7000 LO TRIGGER BIT" %
%   B9:5/10  PT_7000_LO_ALM  "PT-7000 LO ALARM BIT" %
%   B3:0/1  ALARM_RESET  "ALARM RESET" %
%   B9:5/11  PT_7000_LO_ALT  "PT-7000 LO ALERT BIT" %
%   B3:0/0  ALARM_SILENCE  "ALARM SILENCE PUSHBUTTON" %
% Rung: 94 %
SOR GRT N11:23 0 GRT F8:11 F10:23 XIO B3:0/1 BST TON T4:23 1.0 0 0 NXB XIC T4:23/DN OSR B3:6/10 OTE B3:6/11 BND EOR
%   N11:23  PT_7000_HIALM_DLY_SP  "PT-7000 HI ALARM DELAY SP FROM HMI" %
%   F8:11  PT_7000_SCI  "PT-7000 SCALED INPUT" %
%   F10:23  PT_7000_HIALM_SP  "PT-7000 HI ALARM SP" %
%   B3:0/1  ALARM_RESET  "ALARM RESET" %
%   T4:23  PT_7000_HIALM_DLY_TM  "PT-7000 HI ALARM DELAY" %
%   B3:6/10  "OSR" %
%   B3:6/11  "PT-7000 HI TRIGGER BIT" %

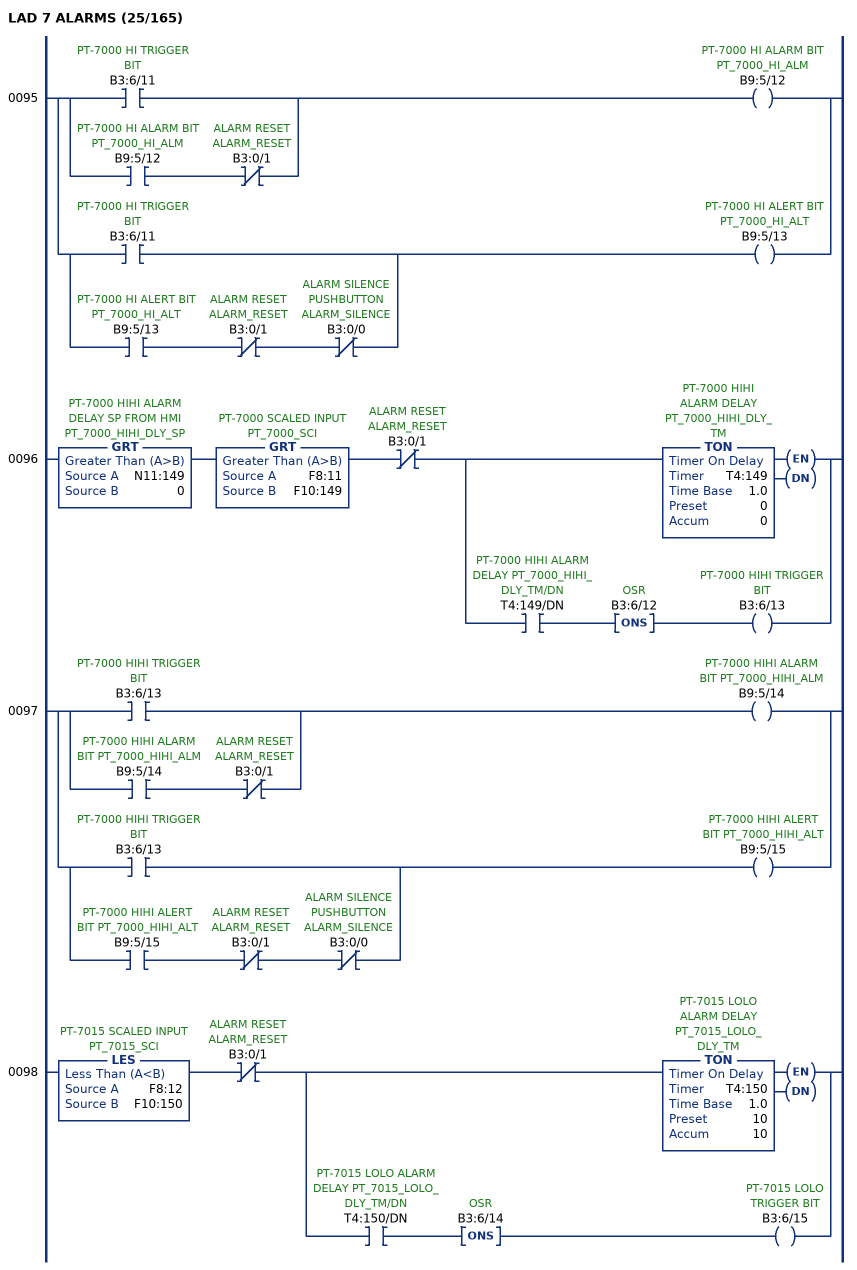
% Rung: 95 %
SOR BST BST XIC B3:6/11 NXB XIC B9:5/12 XIO B3:0/1 BND OTE B9:5/12 NXB BST XIC B3:6/11 NXB XIC B9:5/13 XIO B3:0/1 XIO B3:0/0 BND OTE B9:5/13 BND EOR
%   B3:6/11  "PT-7000 HI TRIGGER BIT" %
%   B9:5/12  PT_7000_HI_ALM  "PT-7000 HI ALARM BIT" %
%   B3:0/1  ALARM_RESET  "ALARM RESET" %
%   B9:5/13  PT_7000_HI_ALT  "PT-7000 HI ALERT BIT" %
%   B3:0/0  ALARM_SILENCE  "ALARM SILENCE PUSHBUTTON" %
% Rung: 96 %
SOR GRT N11:149 0 GRT F8:11 F10:149 XIO B3:0/1 BST TON T4:149 1.0 0 0 NXB XIC T4:149/DN OSR B3:6/12 OTE B3:6/13 BND EOR
%   N11:149  PT_7000_HIHI_DLY_SP  "PT-7000 HIHI ALARM DELAY SP FROM HMI" %
%   F8:11  PT_7000_SCI  "PT-7000 SCALED INPUT" %
%   F10:149  PT_7000_HIHI_SP  "PT-7000 HIHI ALARM SP" %
%   B3:0/1  ALARM_RESET  "ALARM RESET" %
%   T4:149  PT_7000_HIHI_DLY_TM  "PT-7000 HIHI ALARM DELAY" %
%   B3:6/12  "OSR" %
%   B3:6/13  "PT-7000 HIHI TRIGGER BIT" %
% Rung: 97 %
SOR BST BST XIC B3:6/13 NXB XIC B9:5/14 XIO B3:0/1 BND OTE B9:5/14 NXB BST XIC B3:6/13 NXB XIC B9:5/15 XIO B3:0/1 XIO B3:0/0 BND OTE B9:5/15 BND EOR
%   B3:6/13  "PT-7000 HIHI TRIGGER BIT" %
%   B9:5/14  PT_7000_HIHI_ALM  "PT-7000 HIHI ALARM BIT" %
%   B3:0/1  ALARM_RESET  "ALARM RESET" %
%   B9:5/15  PT_7000_HIHI_ALT  "PT-7000 HIHI ALERT BIT" %
%   B3:0/0  ALARM_SILENCE  "ALARM SILENCE PUSHBUTTON" %
% Rung: 98 %
SOR LES F8:12 F10:150 XIO B3:0/1 BST TON T4:150 1.0 10 10 NXB XIC T4:150/DN OSR B3:6/14 OTE B3:6/15 BND EOR
%   F8:12  PT_7015_SCI  "PT-7015 SCALED INPUT" %
%   F10:150  PT_7015_LOLO_SP  "PT-7015 LOLO ALARM SP" %
%   B3:0/1  ALARM_RESET  "ALARM RESET" %
%   T4:150  PT_7015_LOLO_DLY_TM  "PT-7015 LOLO ALARM DELAY" %
%   B3:6/14  "OSR" %
%   B3:6/15  "PT-7015 LOLO TRIGGER BIT" %

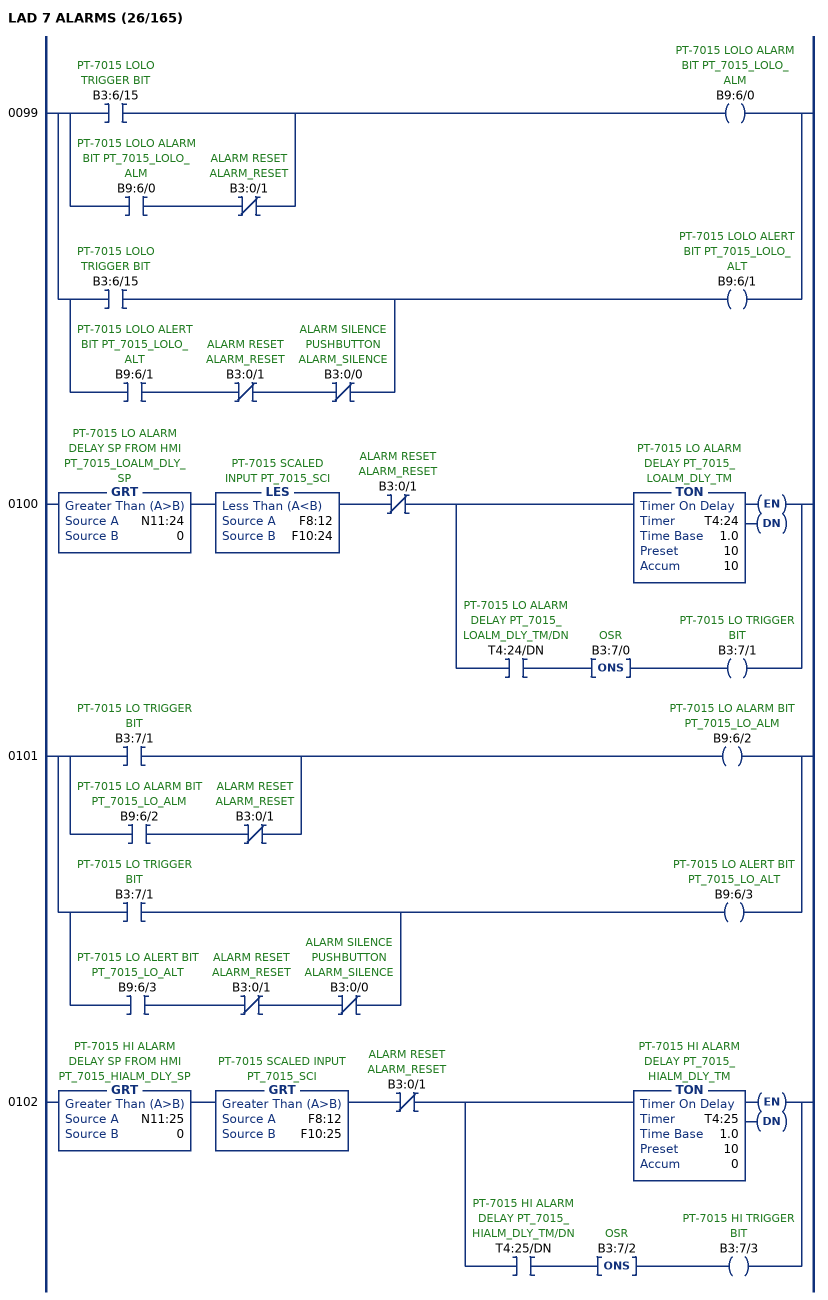
% Rung: 99 %
SOR BST BST XIC B3:6/15 NXB XIC B9:6/0 XIO B3:0/1 BND OTE B9:6/0 NXB BST XIC B3:6/15 NXB XIC B9:6/1 XIO B3:0/1 XIO B3:0/0 BND OTE B9:6/1 BND EOR
%   B3:6/15  "PT-7015 LOLO TRIGGER BIT" %
%   B9:6/0  PT_7015_LOLO_ALM  "PT-7015 LOLO ALARM BIT" %
%   B3:0/1  ALARM_RESET  "ALARM RESET" %
%   B9:6/1  PT_7015_LOLO_ALT  "PT-7015 LOLO ALERT BIT" %
%   B3:0/0  ALARM_SILENCE  "ALARM SILENCE PUSHBUTTON" %
% Rung: 100 %
SOR GRT N11:24 0 LES F8:12 F10:24 XIO B3:0/1 BST TON T4:24 1.0 10 10 NXB XIC T4:24/DN OSR B3:7/0 OTE B3:7/1 BND EOR
%   N11:24  PT_7015_LOALM_DLY_SP  "PT-7015 LO ALARM DELAY SP FROM HMI" %
%   F8:12  PT_7015_SCI  "PT-7015 SCALED INPUT" %
%   F10:24  PT_7015_LOALM_SP  "PT-7015 LO ALARM SP" %
%   B3:0/1  ALARM_RESET  "ALARM RESET" %
%   T4:24  PT_7015_LOALM_DLY_TM  "PT-7015 LO ALARM DELAY" %
%   B3:7/0  "OSR" %
%   B3:7/1  "PT-7015 LO TRIGGER BIT" %
% Rung: 101 %
SOR BST BST XIC B3:7/1 NXB XIC B9:6/2 XIO B3:0/1 BND OTE B9:6/2 NXB BST XIC B3:7/1 NXB XIC B9:6/3 XIO B3:0/1 XIO B3:0/0 BND OTE B9:6/3 BND EOR
%   B3:7/1  "PT-7015 LO TRIGGER BIT" %
%   B9:6/2  PT_7015_LO_ALM  "PT-7015 LO ALARM BIT" %
%   B3:0/1  ALARM_RESET  "ALARM RESET" %
%   B9:6/3  PT_7015_LO_ALT  "PT-7015 LO ALERT BIT" %
%   B3:0/0  ALARM_SILENCE  "ALARM SILENCE PUSHBUTTON" %
% Rung: 102 %
SOR GRT N11:25 0 GRT F8:12 F10:25 XIO B3:0/1 BST TON T4:25 1.0 10 0 NXB XIC T4:25/DN OSR B3:7/2 OTE B3:7/3 BND EOR
%   N11:25  PT_7015_HIALM_DLY_SP  "PT-7015 HI ALARM DELAY SP FROM HMI" %
%   F8:12  PT_7015_SCI  "PT-7015 SCALED INPUT" %
%   F10:25  PT_7015_HIALM_SP  "PT-7015 HI ALARM SP" %
%   B3:0/1  ALARM_RESET  "ALARM RESET" %
%   T4:25  PT_7015_HIALM_DLY_TM  "PT-7015 HI ALARM DELAY" %
%   B3:7/2  "OSR" %
%   B3:7/3  "PT-7015 HI TRIGGER BIT" %

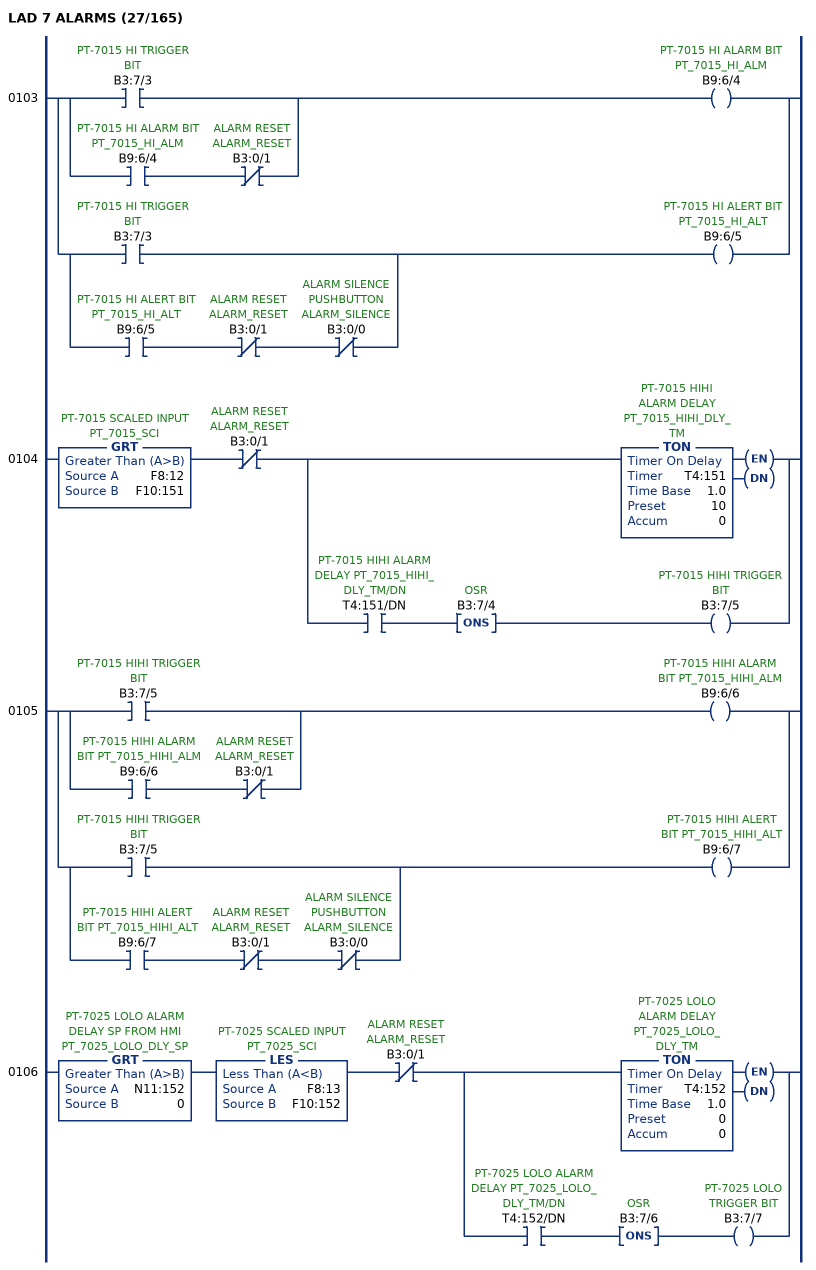
% Rung: 103 %
SOR BST BST XIC B3:7/3 NXB XIC B9:6/4 XIO B3:0/1 BND OTE B9:6/4 NXB BST XIC B3:7/3 NXB XIC B9:6/5 XIO B3:0/1 XIO B3:0/0 BND OTE B9:6/5 BND EOR
%   B3:7/3  "PT-7015 HI TRIGGER BIT" %
%   B9:6/4  PT_7015_HI_ALM  "PT-7015 HI ALARM BIT" %
%   B3:0/1  ALARM_RESET  "ALARM RESET" %
%   B9:6/5  PT_7015_HI_ALT  "PT-7015 HI ALERT BIT" %
%   B3:0/0  ALARM_SILENCE  "ALARM SILENCE PUSHBUTTON" %
% Rung: 104 %
SOR GRT F8:12 F10:151 XIO B3:0/1 BST TON T4:151 1.0 10 0 NXB XIC T4:151/DN OSR B3:7/4 OTE B3:7/5 BND EOR
%   F8:12  PT_7015_SCI  "PT-7015 SCALED INPUT" %
%   F10:151  PT_7015_HIHI_SP  "PT-7015 HIHI ALARM SP" %
%   B3:0/1  ALARM_RESET  "ALARM RESET" %
%   T4:151  PT_7015_HIHI_DLY_TM  "PT-7015 HIHI ALARM DELAY" %
%   B3:7/4  "OSR" %
%   B3:7/5  "PT-7015 HIHI TRIGGER BIT" %
% Rung: 105 %
SOR BST BST XIC B3:7/5 NXB XIC B9:6/6 XIO B3:0/1 BND OTE B9:6/6 NXB BST XIC B3:7/5 NXB XIC B9:6/7 XIO B3:0/1 XIO B3:0/0 BND OTE B9:6/7 BND EOR
%   B3:7/5  "PT-7015 HIHI TRIGGER BIT" %
%   B9:6/6  PT_7015_HIHI_ALM  "PT-7015 HIHI ALARM BIT" %
%   B3:0/1  ALARM_RESET  "ALARM RESET" %
%   B9:6/7  PT_7015_HIHI_ALT  "PT-7015 HIHI ALERT BIT" %
%   B3:0/0  ALARM_SILENCE  "ALARM SILENCE PUSHBUTTON" %
% Rung: 106 %
SOR GRT N11:152 0 LES F8:13 F10:152 XIO B3:0/1 BST TON T4:152 1.0 0 0 NXB XIC T4:152/DN OSR B3:7/6 OTE B3:7/7 BND EOR
%   N11:152  PT_7025_LOLO_DLY_SP  "PT-7025 LOLO ALARM DELAY SP FROM HMI" %
%   F8:13  PT_7025_SCI  "PT-7025 SCALED INPUT" %
%   F10:152  PT_7025_LOLO_SP  "PT-7025 LOLO ALARM SP" %
%   B3:0/1  ALARM_RESET  "ALARM RESET" %
%   T4:152  PT_7025_LOLO_DLY_TM  "PT-7025 LOLO ALARM DELAY" %
%   B3:7/6  "OSR" %
%   B3:7/7  "PT-7025 LOLO TRIGGER BIT" %

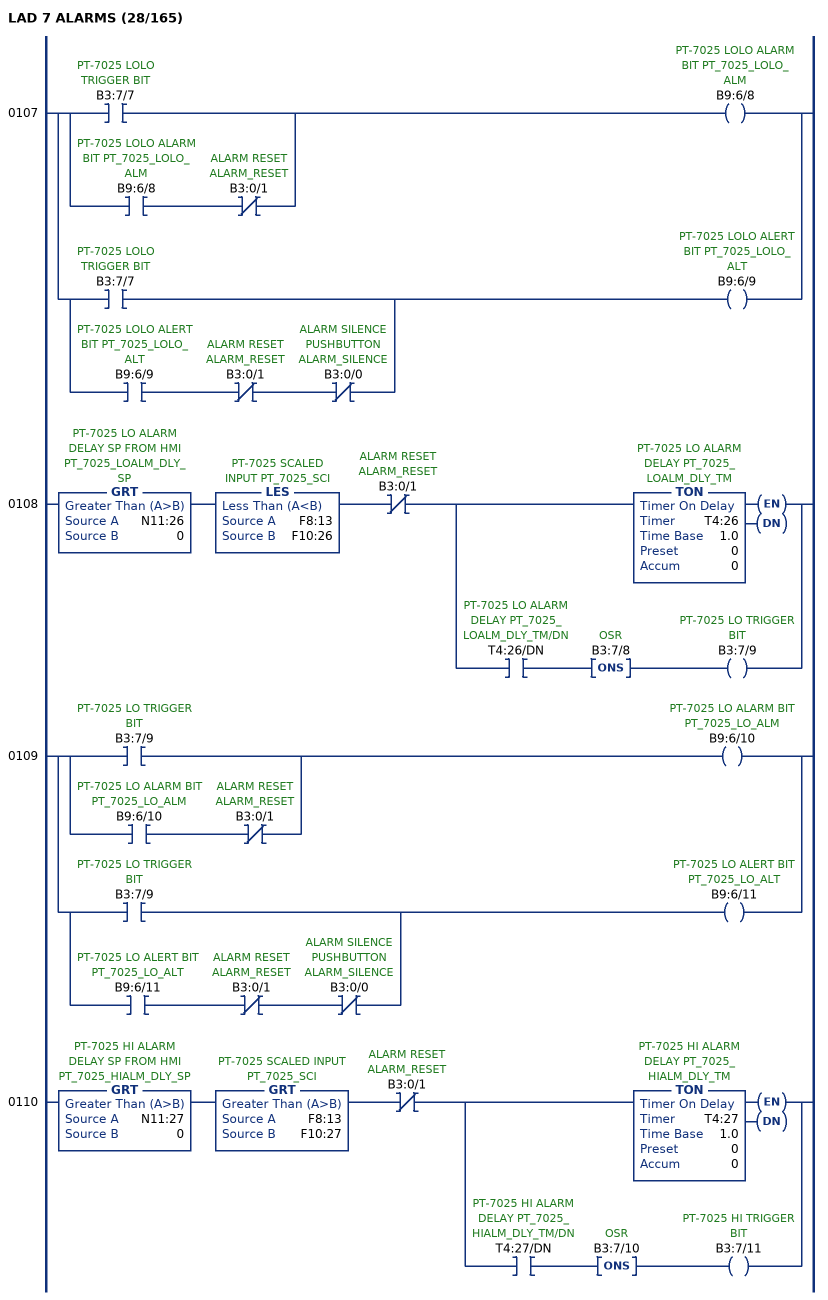
% Rung: 107 %
SOR BST BST XIC B3:7/7 NXB XIC B9:6/8 XIO B3:0/1 BND OTE B9:6/8 NXB BST XIC B3:7/7 NXB XIC B9:6/9 XIO B3:0/1 XIO B3:0/0 BND OTE B9:6/9 BND EOR
%   B3:7/7  "PT-7025 LOLO TRIGGER BIT" %
%   B9:6/8  PT_7025_LOLO_ALM  "PT-7025 LOLO ALARM BIT" %
%   B3:0/1  ALARM_RESET  "ALARM RESET" %
%   B9:6/9  PT_7025_LOLO_ALT  "PT-7025 LOLO ALERT BIT" %
%   B3:0/0  ALARM_SILENCE  "ALARM SILENCE PUSHBUTTON" %
% Rung: 108 %
SOR GRT N11:26 0 LES F8:13 F10:26 XIO B3:0/1 BST TON T4:26 1.0 0 0 NXB XIC T4:26/DN OSR B3:7/8 OTE B3:7/9 BND EOR
%   N11:26  PT_7025_LOALM_DLY_SP  "PT-7025 LO ALARM DELAY SP FROM HMI" %
%   F8:13  PT_7025_SCI  "PT-7025 SCALED INPUT" %
%   F10:26  PT_7025_LOALM_SP  "PT-7025 LO ALARM SP" %
%   B3:0/1  ALARM_RESET  "ALARM RESET" %
%   T4:26  PT_7025_LOALM_DLY_TM  "PT-7025 LO ALARM DELAY" %
%   B3:7/8  "OSR" %
%   B3:7/9  "PT-7025 LO TRIGGER BIT" %
% Rung: 109 %
SOR BST BST XIC B3:7/9 NXB XIC B9:6/10 XIO B3:0/1 BND OTE B9:6/10 NXB BST XIC B3:7/9 NXB XIC B9:6/11 XIO B3:0/1 XIO B3:0/0 BND OTE B9:6/11 BND EOR
%   B3:7/9  "PT-7025 LO TRIGGER BIT" %
%   B9:6/10  PT_7025_LO_ALM  "PT-7025 LO ALARM BIT" %
%   B3:0/1  ALARM_RESET  "ALARM RESET" %
%   B9:6/11  PT_7025_LO_ALT  "PT-7025 LO ALERT BIT" %
%   B3:0/0  ALARM_SILENCE  "ALARM SILENCE PUSHBUTTON" %
% Rung: 110 %
SOR GRT N11:27 0 GRT F8:13 F10:27 XIO B3:0/1 BST TON T4:27 1.0 0 0 NXB XIC T4:27/DN OSR B3:7/10 OTE B3:7/11 BND EOR
%   N11:27  PT_7025_HIALM_DLY_SP  "PT-7025 HI ALARM DELAY SP FROM HMI" %
%   F8:13  PT_7025_SCI  "PT-7025 SCALED INPUT" %
%   F10:27  PT_7025_HIALM_SP  "PT-7025 HI ALARM SP" %
%   B3:0/1  ALARM_RESET  "ALARM RESET" %
%   T4:27  PT_7025_HIALM_DLY_TM  "PT-7025 HI ALARM DELAY" %
%   B3:7/10  "OSR" %
%   B3:7/11  "PT-7025 HI TRIGGER BIT" %

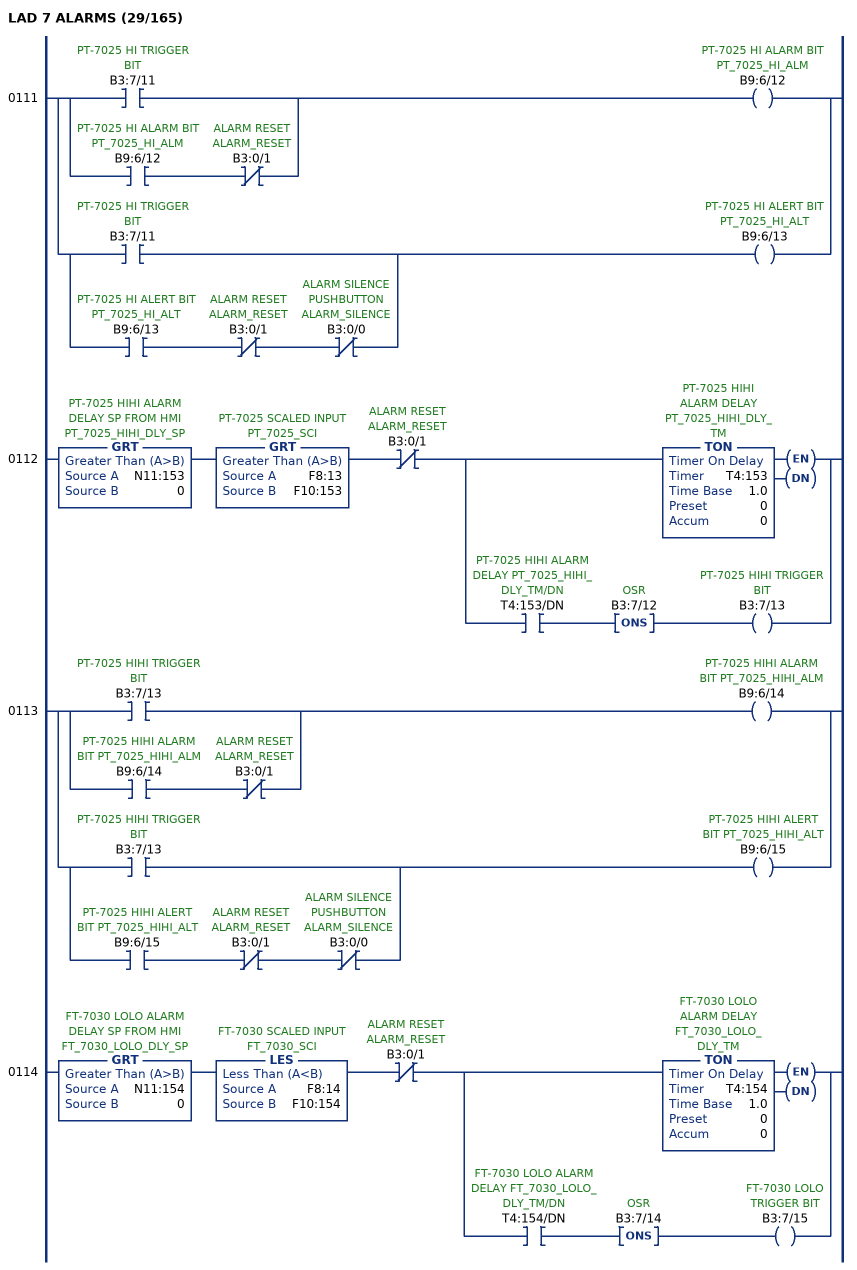
% Rung: 111 %
SOR BST BST XIC B3:7/11 NXB XIC B9:6/12 XIO B3:0/1 BND OTE B9:6/12 NXB BST XIC B3:7/11 NXB XIC B9:6/13 XIO B3:0/1 XIO B3:0/0 BND OTE B9:6/13 BND EOR
%   B3:7/11  "PT-7025 HI TRIGGER BIT" %
%   B9:6/12  PT_7025_HI_ALM  "PT-7025 HI ALARM BIT" %
%   B3:0/1  ALARM_RESET  "ALARM RESET" %
%   B9:6/13  PT_7025_HI_ALT  "PT-7025 HI ALERT BIT" %
%   B3:0/0  ALARM_SILENCE  "ALARM SILENCE PUSHBUTTON" %
% Rung: 112 %
SOR GRT N11:153 0 GRT F8:13 F10:153 XIO B3:0/1 BST TON T4:153 1.0 0 0 NXB XIC T4:153/DN OSR B3:7/12 OTE B3:7/13 BND EOR
%   N11:153  PT_7025_HIHI_DLY_SP  "PT-7025 HIHI ALARM DELAY SP FROM HMI" %
%   F8:13  PT_7025_SCI  "PT-7025 SCALED INPUT" %
%   F10:153  PT_7025_HIHI_SP  "PT-7025 HIHI ALARM SP" %
%   B3:0/1  ALARM_RESET  "ALARM RESET" %
%   T4:153  PT_7025_HIHI_DLY_TM  "PT-7025 HIHI ALARM DELAY" %
%   B3:7/12  "OSR" %
%   B3:7/13  "PT-7025 HIHI TRIGGER BIT" %
% Rung: 113 %
SOR BST BST XIC B3:7/13 NXB XIC B9:6/14 XIO B3:0/1 BND OTE B9:6/14 NXB BST XIC B3:7/13 NXB XIC B9:6/15 XIO B3:0/1 XIO B3:0/0 BND OTE B9:6/15 BND EOR
%   B3:7/13  "PT-7025 HIHI TRIGGER BIT" %
%   B9:6/14  PT_7025_HIHI_ALM  "PT-7025 HIHI ALARM BIT" %
%   B3:0/1  ALARM_RESET  "ALARM RESET" %
%   B9:6/15  PT_7025_HIHI_ALT  "PT-7025 HIHI ALERT BIT" %
%   B3:0/0  ALARM_SILENCE  "ALARM SILENCE PUSHBUTTON" %
% Rung: 114 %
SOR GRT N11:154 0 LES F8:14 F10:154 XIO B3:0/1 BST TON T4:154 1.0 0 0 NXB XIC T4:154/DN OSR B3:7/14 OTE B3:7/15 BND EOR
%   N11:154  FT_7030_LOLO_DLY_SP  "FT-7030 LOLO ALARM DELAY SP FROM HMI" %
%   F8:14  FT_7030_SCI  "FT-7030 SCALED INPUT" %
%   F10:154  FT_7030_LOLO_SP  "FT-7030 LOLO ALARM SP" %
%   B3:0/1  ALARM_RESET  "ALARM RESET" %
%   T4:154  FT_7030_LOLO_DLY_TM  "FT-7030 LOLO ALARM DELAY" %
%   B3:7/14  "OSR" %
%   B3:7/15  "FT-7030 LOLO TRIGGER BIT" %

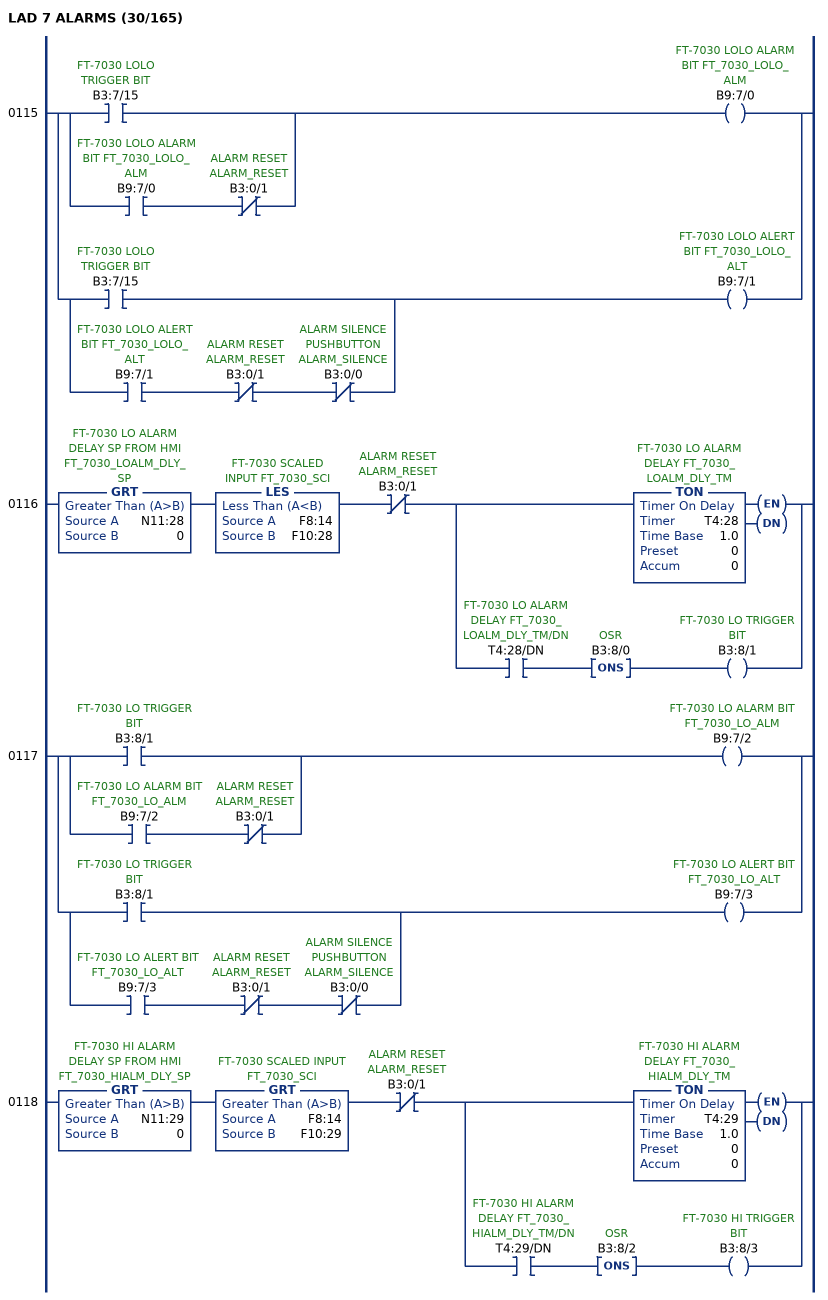
% Rung: 115 %
SOR BST BST XIC B3:7/15 NXB XIC B9:7/0 XIO B3:0/1 BND OTE B9:7/0 NXB BST XIC B3:7/15 NXB XIC B9:7/1 XIO B3:0/1 XIO B3:0/0 BND OTE B9:7/1 BND EOR
%   B3:7/15  "FT-7030 LOLO TRIGGER BIT" %
%   B9:7/0  FT_7030_LOLO_ALM  "FT-7030 LOLO ALARM BIT" %
%   B3:0/1  ALARM_RESET  "ALARM RESET" %
%   B9:7/1  FT_7030_LOLO_ALT  "FT-7030 LOLO ALERT BIT" %
%   B3:0/0  ALARM_SILENCE  "ALARM SILENCE PUSHBUTTON" %
% Rung: 116 %
SOR GRT N11:28 0 LES F8:14 F10:28 XIO B3:0/1 BST TON T4:28 1.0 0 0 NXB XIC T4:28/DN OSR B3:8/0 OTE B3:8/1 BND EOR
%   N11:28  FT_7030_LOALM_DLY_SP  "FT-7030 LO ALARM DELAY SP FROM HMI" %
%   F8:14  FT_7030_SCI  "FT-7030 SCALED INPUT" %
%   F10:28  FT_7030_LOALM_SP  "FT-7030 LO ALARM SP" %
%   B3:0/1  ALARM_RESET  "ALARM RESET" %
%   T4:28  FT_7030_LOALM_DLY_TM  "FT-7030 LO ALARM DELAY" %
%   B3:8/0  "OSR" %
%   B3:8/1  "FT-7030 LO TRIGGER BIT" %
% Rung: 117 %
SOR BST BST XIC B3:8/1 NXB XIC B9:7/2 XIO B3:0/1 BND OTE B9:7/2 NXB BST XIC B3:8/1 NXB XIC B9:7/3 XIO B3:0/1 XIO B3:0/0 BND OTE B9:7/3 BND EOR
%   B3:8/1  "FT-7030 LO TRIGGER BIT" %
%   B9:7/2  FT_7030_LO_ALM  "FT-7030 LO ALARM BIT" %
%   B3:0/1  ALARM_RESET  "ALARM RESET" %
%   B9:7/3  FT_7030_LO_ALT  "FT-7030 LO ALERT BIT" %
%   B3:0/0  ALARM_SILENCE  "ALARM SILENCE PUSHBUTTON" %
% Rung: 118 %
SOR GRT N11:29 0 GRT F8:14 F10:29 XIO B3:0/1 BST TON T4:29 1.0 0 0 NXB XIC T4:29/DN OSR B3:8/2 OTE B3:8/3 BND EOR
%   N11:29  FT_7030_HIALM_DLY_SP  "FT-7030 HI ALARM DELAY SP FROM HMI" %
%   F8:14  FT_7030_SCI  "FT-7030 SCALED INPUT" %
%   F10:29  FT_7030_HIALM_SP  "FT-7030 HI ALARM SP" %
%   B3:0/1  ALARM_RESET  "ALARM RESET" %
%   T4:29  FT_7030_HIALM_DLY_TM  "FT-7030 HI ALARM DELAY" %
%   B3:8/2  "OSR" %
%   B3:8/3  "FT-7030 HI TRIGGER BIT" %

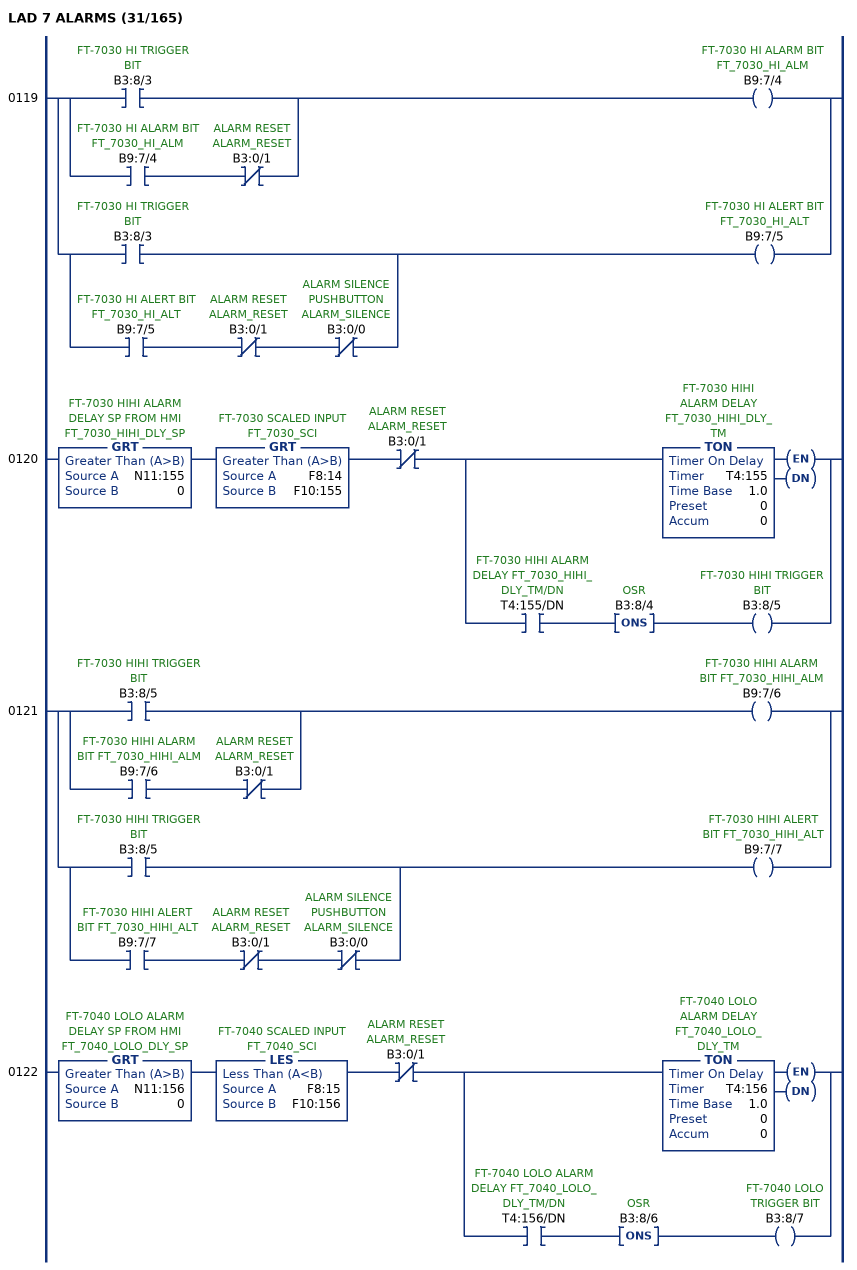
% Rung: 119 %
SOR BST BST XIC B3:8/3 NXB XIC B9:7/4 XIO B3:0/1 BND OTE B9:7/4 NXB BST XIC B3:8/3 NXB XIC B9:7/5 XIO B3:0/1 XIO B3:0/0 BND OTE B9:7/5 BND EOR
%   B3:8/3  "FT-7030 HI TRIGGER BIT" %
%   B9:7/4  FT_7030_HI_ALM  "FT-7030 HI ALARM BIT" %
%   B3:0/1  ALARM_RESET  "ALARM RESET" %
%   B9:7/5  FT_7030_HI_ALT  "FT-7030 HI ALERT BIT" %
%   B3:0/0  ALARM_SILENCE  "ALARM SILENCE PUSHBUTTON" %
% Rung: 120 %
SOR GRT N11:155 0 GRT F8:14 F10:155 XIO B3:0/1 BST TON T4:155 1.0 0 0 NXB XIC T4:155/DN OSR B3:8/4 OTE B3:8/5 BND EOR
%   N11:155  FT_7030_HIHI_DLY_SP  "FT-7030 HIHI ALARM DELAY SP FROM HMI" %
%   F8:14  FT_7030_SCI  "FT-7030 SCALED INPUT" %
%   F10:155  FT_7030_HIHI_SP  "FT-7030 HIHI ALARM SP" %
%   B3:0/1  ALARM_RESET  "ALARM RESET" %
%   T4:155  FT_7030_HIHI_DLY_TM  "FT-7030 HIHI ALARM DELAY" %
%   B3:8/4  "OSR" %
%   B3:8/5  "FT-7030 HIHI TRIGGER BIT" %
% Rung: 121 %
SOR BST BST XIC B3:8/5 NXB XIC B9:7/6 XIO B3:0/1 BND OTE B9:7/6 NXB BST XIC B3:8/5 NXB XIC B9:7/7 XIO B3:0/1 XIO B3:0/0 BND OTE B9:7/7 BND EOR
%   B3:8/5  "FT-7030 HIHI TRIGGER BIT" %
%   B9:7/6  FT_7030_HIHI_ALM  "FT-7030 HIHI ALARM BIT" %
%   B3:0/1  ALARM_RESET  "ALARM RESET" %
%   B9:7/7  FT_7030_HIHI_ALT  "FT-7030 HIHI ALERT BIT" %
%   B3:0/0  ALARM_SILENCE  "ALARM SILENCE PUSHBUTTON" %
% Rung: 122 %
SOR GRT N11:156 0 LES F8:15 F10:156 XIO B3:0/1 BST TON T4:156 1.0 0 0 NXB XIC T4:156/DN OSR B3:8/6 OTE B3:8/7 BND EOR
%   N11:156  FT_7040_LOLO_DLY_SP  "FT-7040 LOLO ALARM DELAY SP FROM HMI" %
%   F8:15  FT_7040_SCI  "FT-7040 SCALED INPUT" %
%   F10:156  FT_7040_LOLO_SP  "FT-7040 LOLO ALARM SP" %
%   B3:0/1  ALARM_RESET  "ALARM RESET" %
%   T4:156  FT_7040_LOLO_DLY_TM  "FT-7040 LOLO ALARM DELAY" %
%   B3:8/6  "OSR" %
%   B3:8/7  "FT-7040 LOLO TRIGGER BIT" %

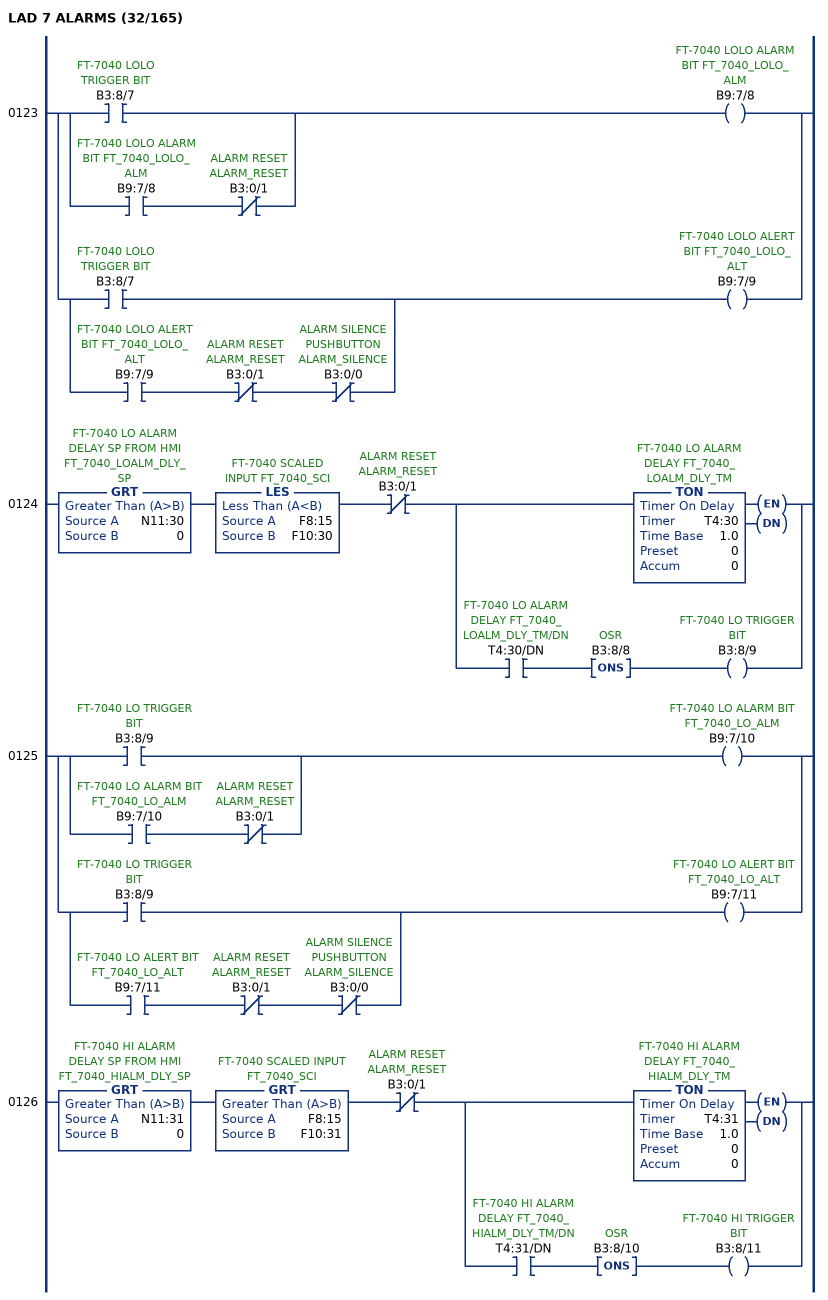
% Rung: 123 %
SOR BST BST XIC B3:8/7 NXB XIC B9:7/8 XIO B3:0/1 BND OTE B9:7/8 NXB BST XIC B3:8/7 NXB XIC B9:7/9 XIO B3:0/1 XIO B3:0/0 BND OTE B9:7/9 BND EOR
%   B3:8/7  "FT-7040 LOLO TRIGGER BIT" %
%   B9:7/8  FT_7040_LOLO_ALM  "FT-7040 LOLO ALARM BIT" %
%   B3:0/1  ALARM_RESET  "ALARM RESET" %
%   B9:7/9  FT_7040_LOLO_ALT  "FT-7040 LOLO ALERT BIT" %
%   B3:0/0  ALARM_SILENCE  "ALARM SILENCE PUSHBUTTON" %
% Rung: 124 %
SOR GRT N11:30 0 LES F8:15 F10:30 XIO B3:0/1 BST TON T4:30 1.0 0 0 NXB XIC T4:30/DN OSR B3:8/8 OTE B3:8/9 BND EOR
%   N11:30  FT_7040_LOALM_DLY_SP  "FT-7040 LO ALARM DELAY SP FROM HMI" %
%   F8:15  FT_7040_SCI  "FT-7040 SCALED INPUT" %
%   F10:30  FT_7040_LOALMSP  "FT-7040 LO ALARM SP" %
%   B3:0/1  ALARM_RESET  "ALARM RESET" %
%   T4:30  FT_7040_LOALM_DLY_TM  "FT-7040 LO ALARM DELAY" %
%   B3:8/8  "OSR" %
%   B3:8/9  "FT-7040 LO TRIGGER BIT" %
% Rung: 125 %
SOR BST BST XIC B3:8/9 NXB XIC B9:7/10 XIO B3:0/1 BND OTE B9:7/10 NXB BST XIC B3:8/9 NXB XIC B9:7/11 XIO B3:0/1 XIO B3:0/0 BND OTE B9:7/11 BND EOR
%   B3:8/9  "FT-7040 LO TRIGGER BIT" %
%   B9:7/10  FT_7040_LO_ALM  "FT-7040 LO ALARM BIT" %
%   B3:0/1  ALARM_RESET  "ALARM RESET" %
%   B9:7/11  FT_7040_LO_ALT  "FT-7040 LO ALERT BIT" %
%   B3:0/0  ALARM_SILENCE  "ALARM SILENCE PUSHBUTTON" %
% Rung: 126 %
SOR GRT N11:31 0 GRT F8:15 F10:31 XIO B3:0/1 BST TON T4:31 1.0 0 0 NXB XIC T4:31/DN OSR B3:8/10 OTE B3:8/11 BND EOR
%   N11:31  FT_7040_HIALM_DLY_SP  "FT-7040 HI ALARM DELAY SP FROM HMI" %
%   F8:15  FT_7040_SCI  "FT-7040 SCALED INPUT" %
%   F10:31  FT_7040_HIALM_SP  "FT-7040 HI ALARM SP" %
%   B3:0/1  ALARM_RESET  "ALARM RESET" %
%   T4:31  FT_7040_HIALM_DLY_TM  "FT-7040 HI ALARM DELAY" %
%   B3:8/10  "OSR" %
%   B3:8/11  "FT-7040 HI TRIGGER BIT" %

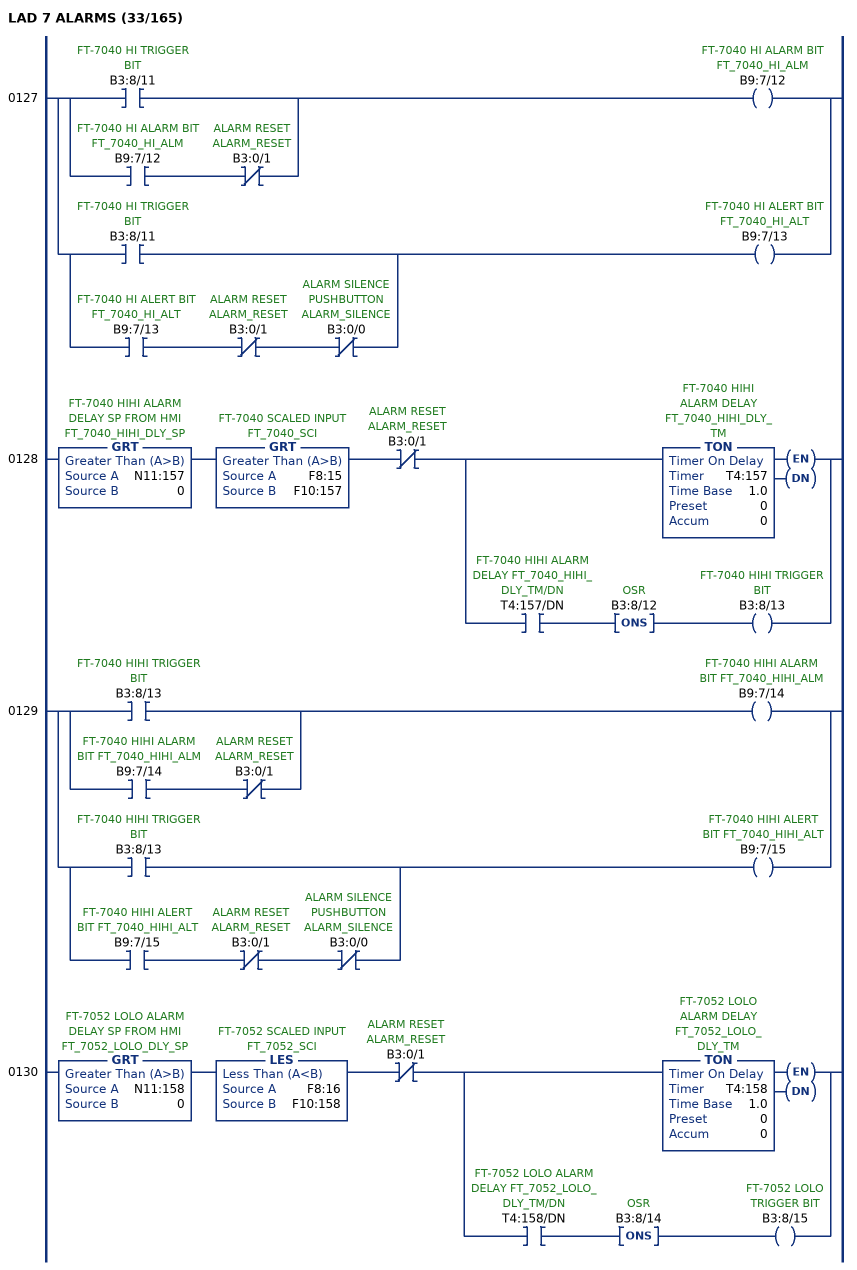
% Rung: 127 %
SOR BST BST XIC B3:8/11 NXB XIC B9:7/12 XIO B3:0/1 BND OTE B9:7/12 NXB BST XIC B3:8/11 NXB XIC B9:7/13 XIO B3:0/1 XIO B3:0/0 BND OTE B9:7/13 BND EOR
%   B3:8/11  "FT-7040 HI TRIGGER BIT" %
%   B9:7/12  FT_7040_HI_ALM  "FT-7040 HI ALARM BIT" %
%   B3:0/1  ALARM_RESET  "ALARM RESET" %
%   B9:7/13  FT_7040_HI_ALT  "FT-7040 HI ALERT BIT" %
%   B3:0/0  ALARM_SILENCE  "ALARM SILENCE PUSHBUTTON" %
% Rung: 128 %
SOR GRT N11:157 0 GRT F8:15 F10:157 XIO B3:0/1 BST TON T4:157 1.0 0 0 NXB XIC T4:157/DN OSR B3:8/12 OTE B3:8/13 BND EOR
%   N11:157  FT_7040_HIHI_DLY_SP  "FT-7040 HIHI ALARM DELAY SP FROM HMI" %
%   F8:15  FT_7040_SCI  "FT-7040 SCALED INPUT" %
%   F10:157  FT_7040_HIHI_SP  "FT-7040 HIHI ALARM SP" %
%   B3:0/1  ALARM_RESET  "ALARM RESET" %
%   T4:157  FT_7040_HIHI_DLY_TM  "FT-7040 HIHI ALARM DELAY" %
%   B3:8/12  "OSR" %
%   B3:8/13  "FT-7040 HIHI TRIGGER BIT" %
% Rung: 129 %
SOR BST BST XIC B3:8/13 NXB XIC B9:7/14 XIO B3:0/1 BND OTE B9:7/14 NXB BST XIC B3:8/13 NXB XIC B9:7/15 XIO B3:0/1 XIO B3:0/0 BND OTE B9:7/15 BND EOR
%   B3:8/13  "FT-7040 HIHI TRIGGER BIT" %
%   B9:7/14  FT_7040_HIHI_ALM  "FT-7040 HIHI ALARM BIT" %
%   B3:0/1  ALARM_RESET  "ALARM RESET" %
%   B9:7/15  FT_7040_HIHI_ALT  "FT-7040 HIHI ALERT BIT" %
%   B3:0/0  ALARM_SILENCE  "ALARM SILENCE PUSHBUTTON" %
% Rung: 130 %
SOR GRT N11:158 0 LES F8:16 F10:158 XIO B3:0/1 BST TON T4:158 1.0 0 0 NXB XIC T4:158/DN OSR B3:8/14 OTE B3:8/15 BND EOR
%   N11:158  FT_7052_LOLO_DLY_SP  "FT-7052 LOLO ALARM DELAY SP FROM HMI" %
%   F8:16  FT_7052_SCI  "FT-7052 SCALED INPUT" %
%   F10:158  FT_7052_LOLO_SP  "FT-7052 LOLO ALARM SP" %
%   B3:0/1  ALARM_RESET  "ALARM RESET" %
%   T4:158  FT_7052_LOLO_DLY_TM  "FT-7052 LOLO ALARM DELAY" %
%   B3:8/14  "OSR" %
%   B3:8/15  "FT-7052 LOLO TRIGGER BIT" %

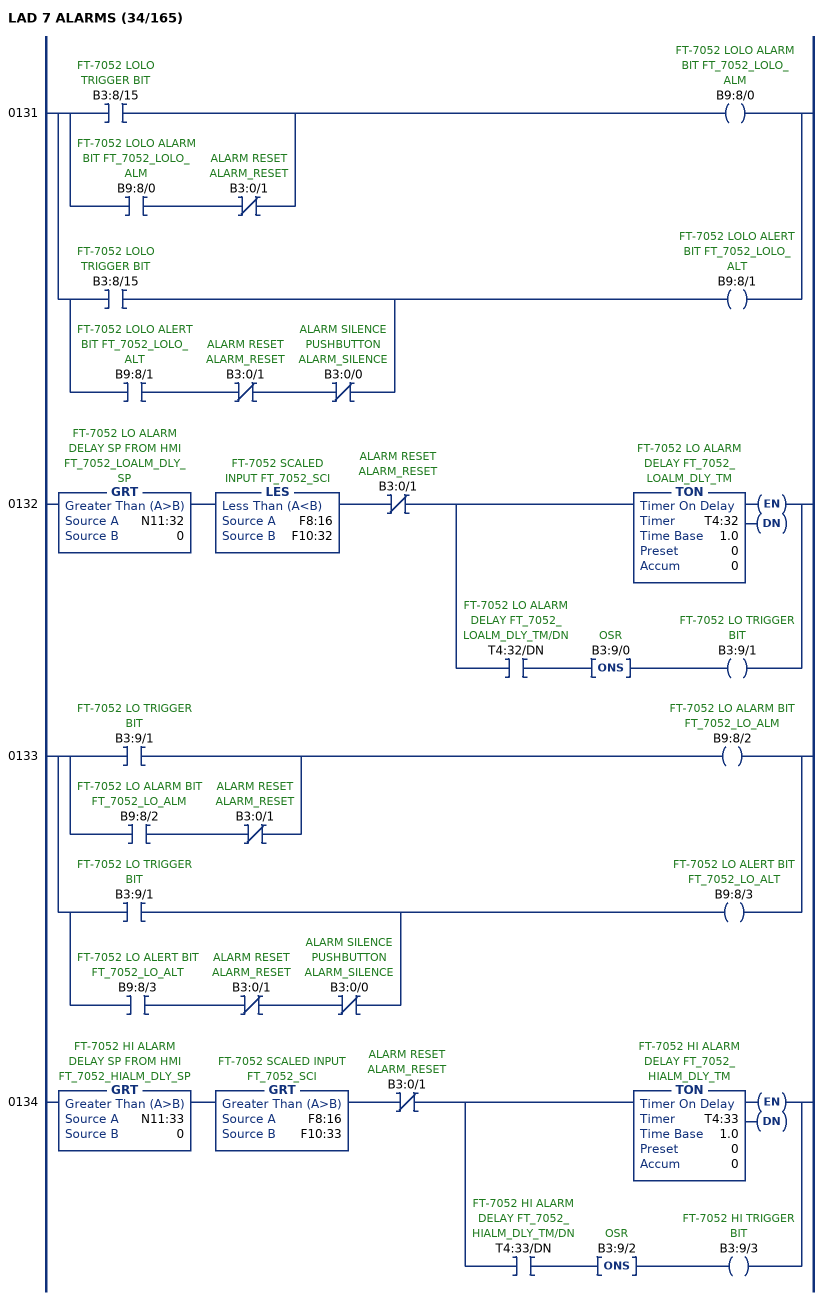
% Rung: 131 %
SOR BST BST XIC B3:8/15 NXB XIC B9:8/0 XIO B3:0/1 BND OTE B9:8/0 NXB BST XIC B3:8/15 NXB XIC B9:8/1 XIO B3:0/1 XIO B3:0/0 BND OTE B9:8/1 BND EOR
%   B3:8/15  "FT-7052 LOLO TRIGGER BIT" %
%   B9:8/0  FT_7052_LOLO_ALM  "FT-7052 LOLO ALARM BIT" %
%   B3:0/1  ALARM_RESET  "ALARM RESET" %
%   B9:8/1  FT_7052_LOLO_ALT  "FT-7052 LOLO ALERT BIT" %
%   B3:0/0  ALARM_SILENCE  "ALARM SILENCE PUSHBUTTON" %
% Rung: 132 %
SOR GRT N11:32 0 LES F8:16 F10:32 XIO B3:0/1 BST TON T4:32 1.0 0 0 NXB XIC T4:32/DN OSR B3:9/0 OTE B3:9/1 BND EOR
%   N11:32  FT_7052_LOALM_DLY_SP  "FT-7052 LO ALARM DELAY SP FROM HMI" %
%   F8:16  FT_7052_SCI  "FT-7052 SCALED INPUT" %
%   F10:32  FT_7052_LOALM_SP  "FT-7052 LO ALARM SP" %
%   B3:0/1  ALARM_RESET  "ALARM RESET" %
%   T4:32  FT_7052_LOALM_DLY_TM  "FT-7052 LO ALARM DELAY" %
%   B3:9/0  "OSR" %
%   B3:9/1  "FT-7052 LO TRIGGER BIT" %
% Rung: 133 %
SOR BST BST XIC B3:9/1 NXB XIC B9:8/2 XIO B3:0/1 BND OTE B9:8/2 NXB BST XIC B3:9/1 NXB XIC B9:8/3 XIO B3:0/1 XIO B3:0/0 BND OTE B9:8/3 BND EOR
%   B3:9/1  "FT-7052 LO TRIGGER BIT" %
%   B9:8/2  FT_7052_LO_ALM  "FT-7052 LO ALARM BIT" %
%   B3:0/1  ALARM_RESET  "ALARM RESET" %
%   B9:8/3  FT_7052_LO_ALT  "FT-7052 LO ALERT BIT" %
%   B3:0/0  ALARM_SILENCE  "ALARM SILENCE PUSHBUTTON" %
% Rung: 134 %
SOR GRT N11:33 0 GRT F8:16 F10:33 XIO B3:0/1 BST TON T4:33 1.0 0 0 NXB XIC T4:33/DN OSR B3:9/2 OTE B3:9/3 BND EOR
%   N11:33  FT_7052_HIALM_DLY_SP  "FT-7052 HI ALARM DELAY SP FROM HMI" %
%   F8:16  FT_7052_SCI  "FT-7052 SCALED INPUT" %
%   F10:33  FT_7052_HIALM_SP  "FT-7052 HI ALARM SP" %
%   B3:0/1  ALARM_RESET  "ALARM RESET" %
%   T4:33  FT_7052_HIALM_DLY_TM  "FT-7052 HI ALARM DELAY" %
%   B3:9/2  "OSR" %
%   B3:9/3  "FT-7052 HI TRIGGER BIT" %

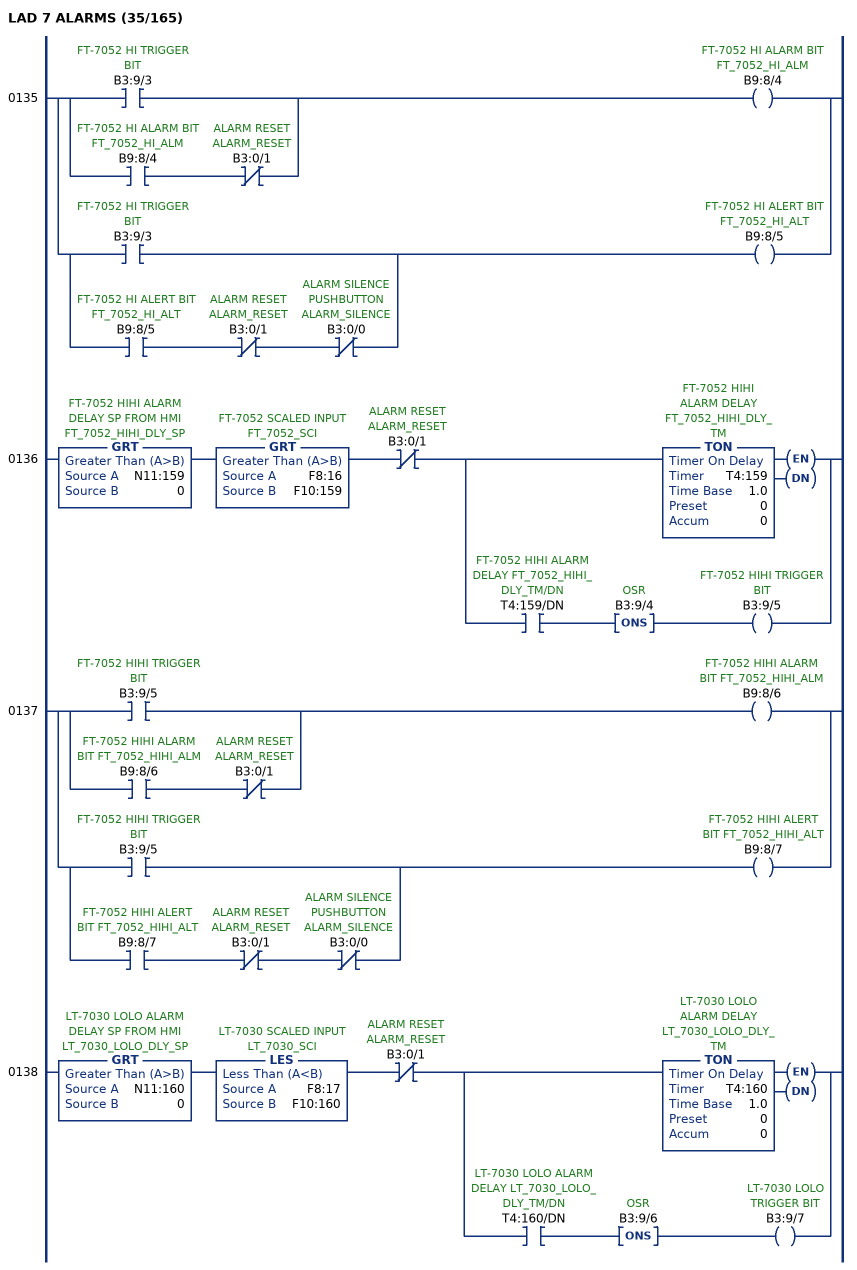
% Rung: 135 %
SOR BST BST XIC B3:9/3 NXB XIC B9:8/4 XIO B3:0/1 BND OTE B9:8/4 NXB BST XIC B3:9/3 NXB XIC B9:8/5 XIO B3:0/1 XIO B3:0/0 BND OTE B9:8/5 BND EOR
%   B3:9/3  "FT-7052 HI TRIGGER BIT" %
%   B9:8/4  FT_7052_HI_ALM  "FT-7052 HI ALARM BIT" %
%   B3:0/1  ALARM_RESET  "ALARM RESET" %
%   B9:8/5  FT_7052_HI_ALT  "FT-7052 HI ALERT BIT" %
%   B3:0/0  ALARM_SILENCE  "ALARM SILENCE PUSHBUTTON" %
% Rung: 136 %
SOR GRT N11:159 0 GRT F8:16 F10:159 XIO B3:0/1 BST TON T4:159 1.0 0 0 NXB XIC T4:159/DN OSR B3:9/4 OTE B3:9/5 BND EOR
%   N11:159  FT_7052_HIHI_DLY_SP  "FT-7052 HIHI ALARM DELAY SP FROM HMI" %
%   F8:16  FT_7052_SCI  "FT-7052 SCALED INPUT" %
%   F10:159  FT_7052_HIHI_SP  "FT-7052 HIHI ALARM SP" %
%   B3:0/1  ALARM_RESET  "ALARM RESET" %
%   T4:159  FT_7052_HIHI_DLY_TM  "FT-7052 HIHI ALARM DELAY" %
%   B3:9/4  "OSR" %
%   B3:9/5  "FT-7052 HIHI TRIGGER BIT" %
% Rung: 137 %
SOR BST BST XIC B3:9/5 NXB XIC B9:8/6 XIO B3:0/1 BND OTE B9:8/6 NXB BST XIC B3:9/5 NXB XIC B9:8/7 XIO B3:0/1 XIO B3:0/0 BND OTE B9:8/7 BND EOR
%   B3:9/5  "FT-7052 HIHI TRIGGER BIT" %
%   B9:8/6  FT_7052_HIHI_ALM  "FT-7052 HIHI ALARM BIT" %
%   B3:0/1  ALARM_RESET  "ALARM RESET" %
%   B9:8/7  FT_7052_HIHI_ALT  "FT-7052 HIHI ALERT BIT" %
%   B3:0/0  ALARM_SILENCE  "ALARM SILENCE PUSHBUTTON" %
% Rung: 138 %
SOR GRT N11:160 0 LES F8:17 F10:160 XIO B3:0/1 BST TON T4:160 1.0 0 0 NXB XIC T4:160/DN OSR B3:9/6 OTE B3:9/7 BND EOR
%   N11:160  LT_7030_LOLO_DLY_SP  "LT-7030 LOLO ALARM DELAY SP FROM HMI" %
%   F8:17  LT_7030_SCI  "LT-7030 SCALED INPUT" %
%   F10:160  LT_7030_LOLO_SP  "LT-7030 LOLO ALARM SP" %
%   B3:0/1  ALARM_RESET  "ALARM RESET" %
%   T4:160  LT_7030_LOLO_DLY_TM  "LT-7030 LOLO ALARM DELAY" %
%   B3:9/6  "OSR" %
%   B3:9/7  "LT-7030 LOLO TRIGGER BIT" %

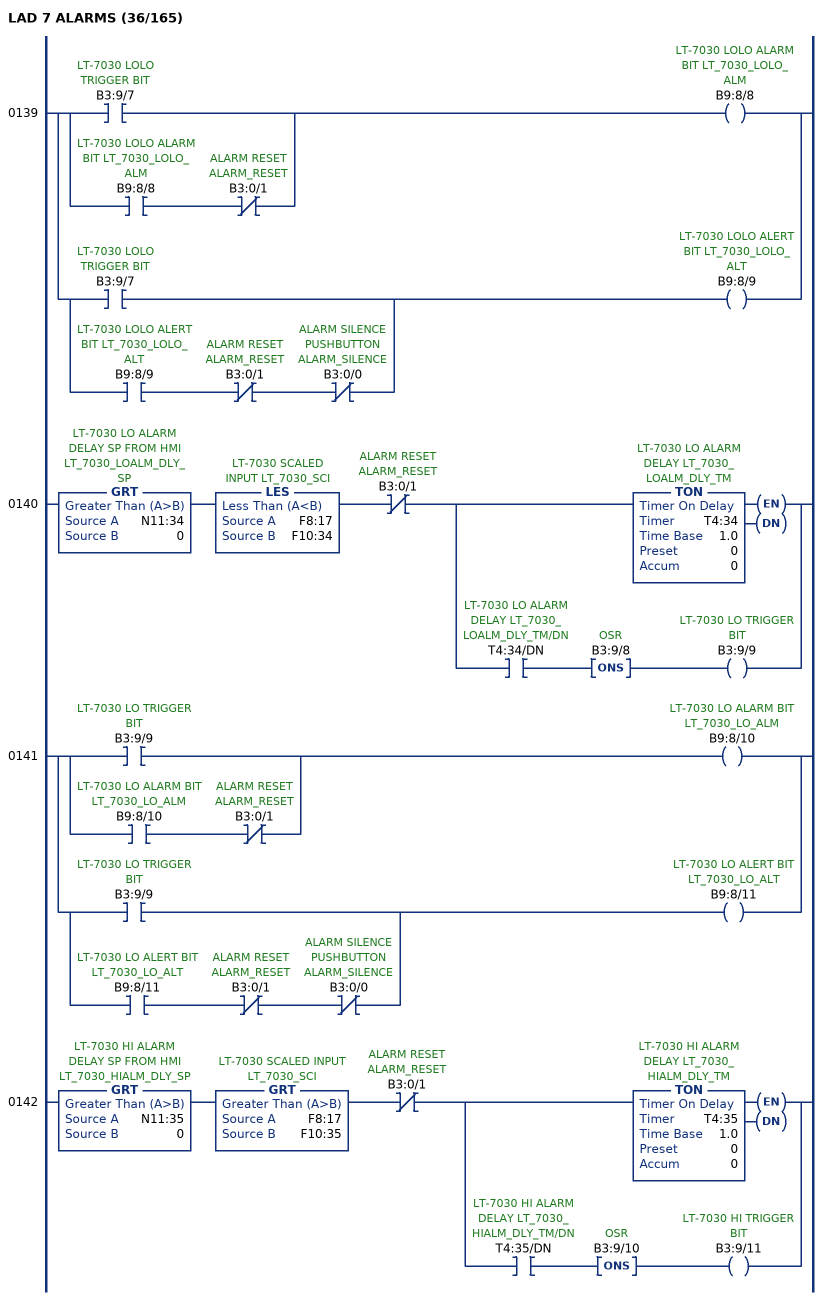
% Rung: 139 %
SOR BST BST XIC B3:9/7 NXB XIC B9:8/8 XIO B3:0/1 BND OTE B9:8/8 NXB BST XIC B3:9/7 NXB XIC B9:8/9 XIO B3:0/1 XIO B3:0/0 BND OTE B9:8/9 BND EOR
%   B3:9/7  "LT-7030 LOLO TRIGGER BIT" %
%   B9:8/8  LT_7030_LOLO_ALM  "LT-7030 LOLO ALARM BIT" %
%   B3:0/1  ALARM_RESET  "ALARM RESET" %
%   B9:8/9  LT_7030_LOLO_ALT  "LT-7030 LOLO ALERT BIT" %
%   B3:0/0  ALARM_SILENCE  "ALARM SILENCE PUSHBUTTON" %
% Rung: 140 %
SOR GRT N11:34 0 LES F8:17 F10:34 XIO B3:0/1 BST TON T4:34 1.0 0 0 NXB XIC T4:34/DN OSR B3:9/8 OTE B3:9/9 BND EOR
%   N11:34  LT_7030_LOALM_DLY_SP  "LT-7030 LO ALARM DELAY SP FROM HMI" %
%   F8:17  LT_7030_SCI  "LT-7030 SCALED INPUT" %
%   F10:34  LT_7030_LOALM_SP  "LT-7030 LO ALARM SP" %
%   B3:0/1  ALARM_RESET  "ALARM RESET" %
%   T4:34  LT_7030_LOALM_DLY_TM  "LT-7030 LO ALARM DELAY" %
%   B3:9/8  "OSR" %
%   B3:9/9  "LT-7030 LO TRIGGER BIT" %
% Rung: 141 %
SOR BST BST XIC B3:9/9 NXB XIC B9:8/10 XIO B3:0/1 BND OTE B9:8/10 NXB BST XIC B3:9/9 NXB XIC B9:8/11 XIO B3:0/1 XIO B3:0/0 BND OTE B9:8/11 BND EOR
%   B3:9/9  "LT-7030 LO TRIGGER BIT" %
%   B9:8/10  LT_7030_LO_ALM  "LT-7030 LO ALARM BIT" %
%   B3:0/1  ALARM_RESET  "ALARM RESET" %
%   B9:8/11  LT_7030_LO_ALT  "LT-7030 LO ALERT BIT" %
%   B3:0/0  ALARM_SILENCE  "ALARM SILENCE PUSHBUTTON" %
% Rung: 142 %
SOR GRT N11:35 0 GRT F8:17 F10:35 XIO B3:0/1 BST TON T4:35 1.0 0 0 NXB XIC T4:35/DN OSR B3:9/10 OTE B3:9/11 BND EOR
%   N11:35  LT_7030_HIALM_DLY_SP  "LT-7030 HI ALARM DELAY SP FROM HMI" %
%   F8:17  LT_7030_SCI  "LT-7030 SCALED INPUT" %
%   F10:35  LT_7030_HIALM_SP  "LT-7030 HI ALARM SP" %
%   B3:0/1  ALARM_RESET  "ALARM RESET" %
%   T4:35  LT_7030_HIALM_DLY_TM  "LT-7030 HI ALARM DELAY" %
%   B3:9/10  "OSR" %
%   B3:9/11  "LT-7030 HI TRIGGER BIT" %

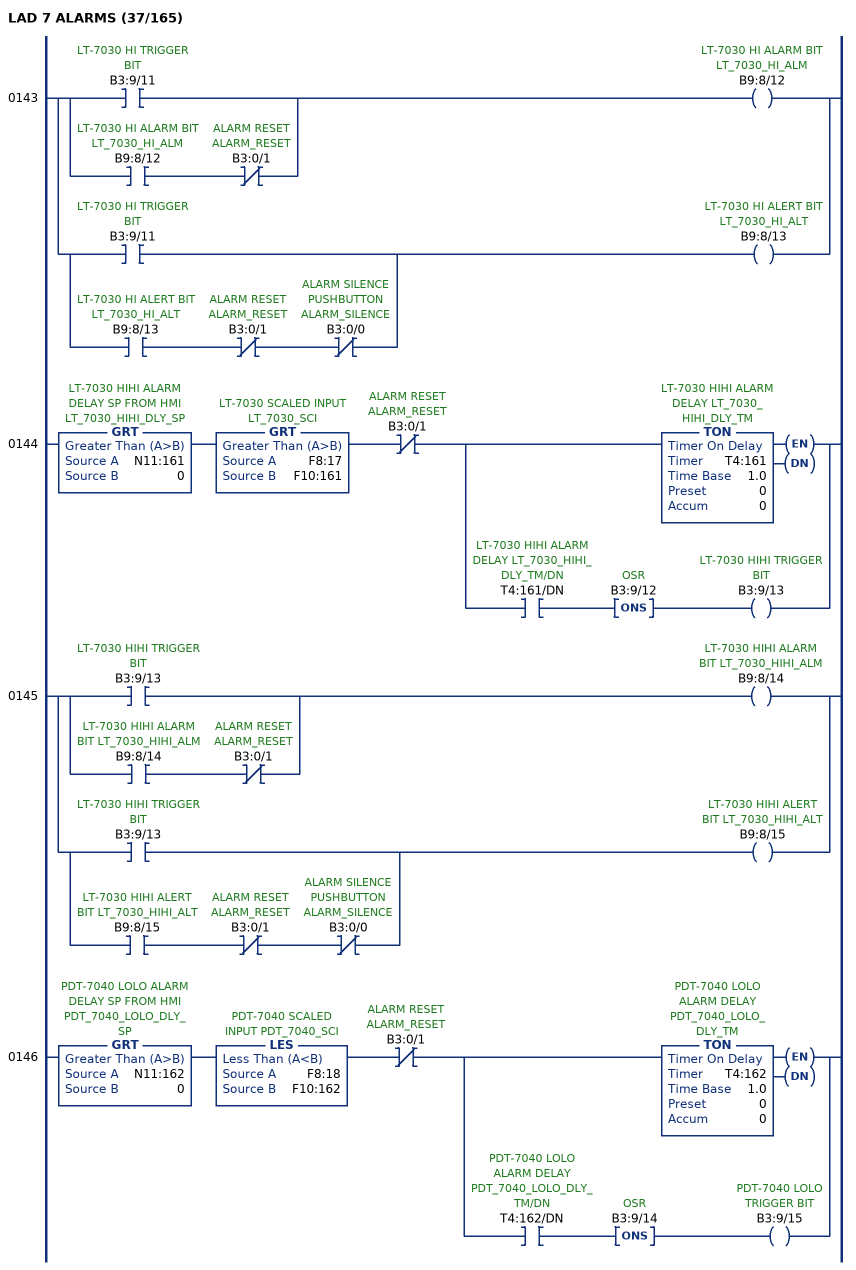
% Rung: 143 %
SOR BST BST XIC B3:9/11 NXB XIC B9:8/12 XIO B3:0/1 BND OTE B9:8/12 NXB BST XIC B3:9/11 NXB XIC B9:8/13 XIO B3:0/1 XIO B3:0/0 BND OTE B9:8/13 BND EOR
%   B3:9/11  "LT-7030 HI TRIGGER BIT" %
%   B9:8/12  LT_7030_HI_ALM  "LT-7030 HI ALARM BIT" %
%   B3:0/1  ALARM_RESET  "ALARM RESET" %
%   B9:8/13  LT_7030_HI_ALT  "LT-7030 HI ALERT BIT" %
%   B3:0/0  ALARM_SILENCE  "ALARM SILENCE PUSHBUTTON" %
% Rung: 144 %
SOR GRT N11:161 0 GRT F8:17 F10:161 XIO B3:0/1 BST TON T4:161 1.0 0 0 NXB XIC T4:161/DN OSR B3:9/12 OTE B3:9/13 BND EOR
%   N11:161  LT_7030_HIHI_DLY_SP  "LT-7030 HIHI ALARM DELAY SP FROM HMI" %
%   F8:17  LT_7030_SCI  "LT-7030 SCALED INPUT" %
%   F10:161  LT_7030_HIHI_SP  "LT-7030 HIHI ALARM SP" %
%   B3:0/1  ALARM_RESET  "ALARM RESET" %
%   T4:161  LT_7030_HIHI_DLY_TM  "LT-7030 HIHI ALARM DELAY" %
%   B3:9/12  "OSR" %
%   B3:9/13  "LT-7030 HIHI TRIGGER BIT" %
% Rung: 145 %
SOR BST BST XIC B3:9/13 NXB XIC B9:8/14 XIO B3:0/1 BND OTE B9:8/14 NXB BST XIC B3:9/13 NXB XIC B9:8/15 XIO B3:0/1 XIO B3:0/0 BND OTE B9:8/15 BND EOR
%   B3:9/13  "LT-7030 HIHI TRIGGER BIT" %
%   B9:8/14  LT_7030_HIHI_ALM  "LT-7030 HIHI ALARM BIT" %
%   B3:0/1  ALARM_RESET  "ALARM RESET" %
%   B9:8/15  LT_7030_HIHI_ALT  "LT-7030 HIHI ALERT BIT" %
%   B3:0/0  ALARM_SILENCE  "ALARM SILENCE PUSHBUTTON" %
% Rung: 146 %
SOR GRT N11:162 0 LES F8:18 F10:162 XIO B3:0/1 BST TON T4:162 1.0 0 0 NXB XIC T4:162/DN OSR B3:9/14 OTE B3:9/15 BND EOR
%   N11:162  PDT_7040_LOLO_DLY_SP  "PDT-7040 LOLO ALARM DELAY SP FROM HMI" %
%   F8:18  PDT_7040_SCI  "PDT-7040 SCALED INPUT" %
%   F10:162  PDT_7040_LOLO_SP  "PDT-7040 LOLO ALARM SP" %
%   B3:0/1  ALARM_RESET  "ALARM RESET" %
%   T4:162  PDT_7040_LOLO_DLY_TM  "PDT-7040 LOLO ALARM DELAY" %
%   B3:9/14  "OSR" %
%   B3:9/15  "PDT-7040 LOLO TRIGGER BIT" %

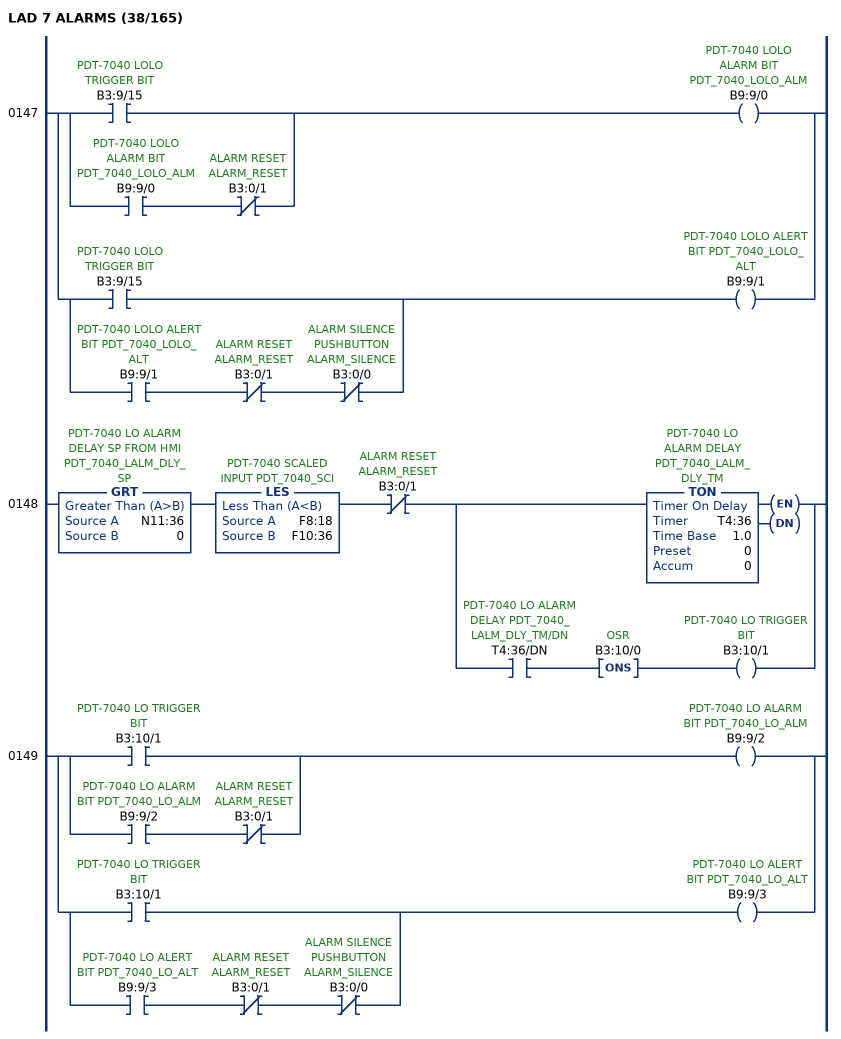
% Rung: 147 %
SOR BST BST XIC B3:9/15 NXB XIC B9:9/0 XIO B3:0/1 BND OTE B9:9/0 NXB BST XIC B3:9/15 NXB XIC B9:9/1 XIO B3:0/1 XIO B3:0/0 BND OTE B9:9/1 BND EOR
%   B3:9/15  "PDT-7040 LOLO TRIGGER BIT" %
%   B9:9/0  PDT_7040_LOLO_ALM  "PDT-7040 LOLO ALARM BIT" %
%   B3:0/1  ALARM_RESET  "ALARM RESET" %
%   B9:9/1  PDT_7040_LOLO_ALT  "PDT-7040 LOLO ALERT BIT" %
%   B3:0/0  ALARM_SILENCE  "ALARM SILENCE PUSHBUTTON" %
% Rung: 148 %
SOR GRT N11:36 0 LES F8:18 F10:36 XIO B3:0/1 BST TON T4:36 1.0 0 0 NXB XIC T4:36/DN OSR B3:10/0 OTE B3:10/1 BND EOR
%   N11:36  PDT_7040_LALM_DLY_SP  "PDT-7040 LO ALARM DELAY SP FROM HMI" %
%   F8:18  PDT_7040_SCI  "PDT-7040 SCALED INPUT" %
%   F10:36  PDT_7040_LOALM_SP  "PDT-7040 LO ALARM SP" %
%   B3:0/1  ALARM_RESET  "ALARM RESET" %
%   T4:36  PDT_7040_LALM_DLY_TM  "PDT-7040 LO ALARM DELAY" %
%   B3:10/0  "OSR" %
%   B3:10/1  "PDT-7040 LO TRIGGER BIT" %
% Rung: 149 %
SOR BST BST XIC B3:10/1 NXB XIC B9:9/2 XIO B3:0/1 BND OTE B9:9/2 NXB BST XIC B3:10/1 NXB XIC B9:9/3 XIO B3:0/1 XIO B3:0/0 BND OTE B9:9/3 BND EOR
%   B3:10/1  "PDT-7040 LO TRIGGER BIT" %
%   B9:9/2  PDT_7040_LO_ALM  "PDT-7040 LO ALARM BIT" %
%   B3:0/1  ALARM_RESET  "ALARM RESET" %
%   B9:9/3  PDT_7040_LO_ALT  "PDT-7040 LO ALERT BIT" %
%   B3:0/0  ALARM_SILENCE  "ALARM SILENCE PUSHBUTTON" %

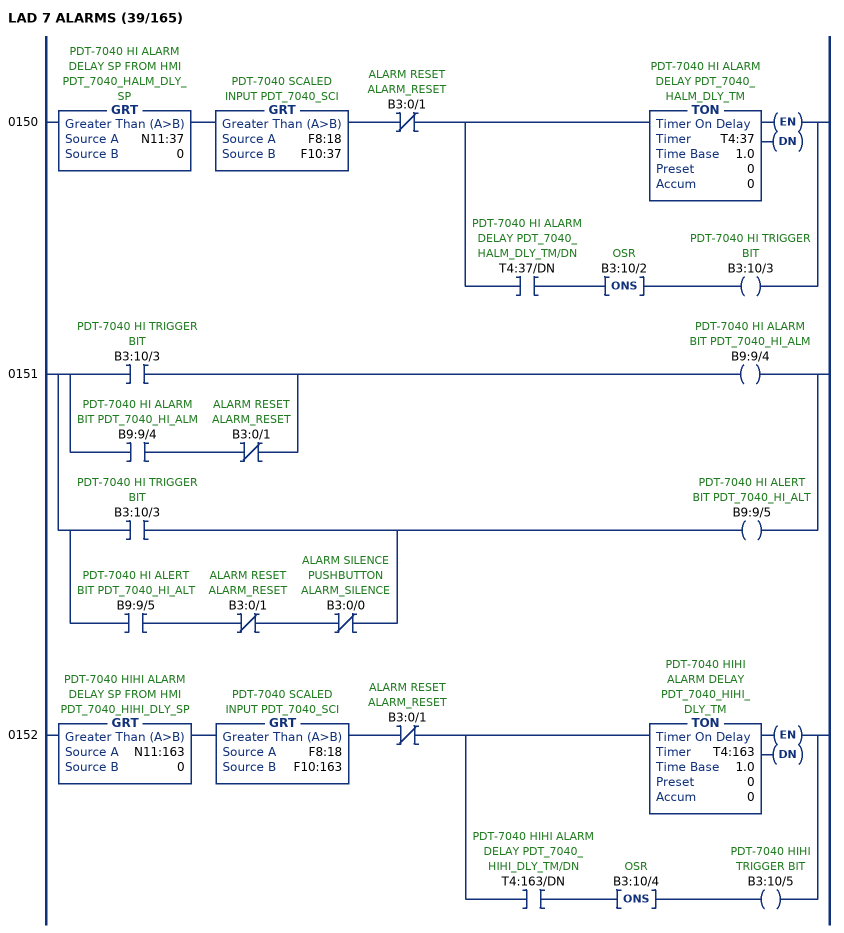
% Rung: 150 %
SOR GRT N11:37 0 GRT F8:18 F10:37 XIO B3:0/1 BST TON T4:37 1.0 0 0 NXB XIC T4:37/DN OSR B3:10/2 OTE B3:10/3 BND EOR
%   N11:37  PDT_7040_HALM_DLY_SP  "PDT-7040 HI ALARM DELAY SP FROM HMI" %
%   F8:18  PDT_7040_SCI  "PDT-7040 SCALED INPUT" %
%   F10:37  PDT_7040_HIALM_SP  "PDT-7040 HI ALARM SP" %
%   B3:0/1  ALARM_RESET  "ALARM RESET" %
%   T4:37  PDT_7040_HALM_DLY_TM  "PDT-7040 HI ALARM DELAY" %
%   B3:10/2  "OSR" %
%   B3:10/3  "PDT-7040 HI TRIGGER BIT" %
% Rung: 151 %
SOR BST BST XIC B3:10/3 NXB XIC B9:9/4 XIO B3:0/1 BND OTE B9:9/4 NXB BST XIC B3:10/3 NXB XIC B9:9/5 XIO B3:0/1 XIO B3:0/0 BND OTE B9:9/5 BND EOR
%   B3:10/3  "PDT-7040 HI TRIGGER BIT" %
%   B9:9/4  PDT_7040_HI_ALM  "PDT-7040 HI ALARM BIT" %
%   B3:0/1  ALARM_RESET  "ALARM RESET" %
%   B9:9/5  PDT_7040_HI_ALT  "PDT-7040 HI ALERT BIT" %
%   B3:0/0  ALARM_SILENCE  "ALARM SILENCE PUSHBUTTON" %
% Rung: 152 %
SOR GRT N11:163 0 GRT F8:18 F10:163 XIO B3:0/1 BST TON T4:163 1.0 0 0 NXB XIC T4:163/DN OSR B3:10/4 OTE B3:10/5 BND EOR
%   N11:163  PDT_7040_HIHI_DLY_SP  "PDT-7040 HIHI ALARM DELAY SP FROM HMI" %
%   F8:18  PDT_7040_SCI  "PDT-7040 SCALED INPUT" %
%   F10:163  PDT_7040_HIHI_SP  "PDT-7040 HIHI ALARM SP" %
%   B3:0/1  ALARM_RESET  "ALARM RESET" %
%   T4:163  PDT_7040_HIHI_DLY_TM  "PDT-7040 HIHI ALARM DELAY" %
%   B3:10/4  "OSR" %
%   B3:10/5  "PDT-7040 HIHI TRIGGER BIT" %

